SPLINE
SPL {X  -140.879, Y  +291.363, Z    +0.000, E1   +48.273, E3 +172222.912}
SPL {X  -158.845, Y  +331.507, Z    +0.000, E1   +33.834, E3 +172232.246}
SPL {X  -164.164, Y  +356.358, Z    +0.000, E1   +18.707, E3 +172228.569}
SPL {X  -165.341, Y  +368.384, Z    +0.000, E1   +10.076, E3 +172229.313}
SPL {X  -165.648, Y  +377.641, Z    +0.000, E1    +2.653, E3 +172228.664}
SPL {X  -165.650, Y  +380.939, Z    +0.000, E1    -0.407, E3 +172227.475}
SPL {X  -165.650, Y  +384.595, Z    +0.000, E1    -6.546, E3 +172226.958}
SPL {X  -165.650, Y  +389.276, Z    +0.000, E1   -15.245, E3 +172226.466}
SPL {X  -165.650, Y  +395.801, Z    +0.000, E1   -28.236, E3 +172226.094}
SPL {X  -165.650, Y  +403.802, Z    +0.000, E1   -41.748, E3 +172225.915}
SPL {X  -165.650, Y  +419.045, Z    +0.000, E1   -60.641, E3 +172223.236}
SPL {X  -165.650, Y  +474.102, Z    +0.000, E1   -73.446, E3 +172235.019}
SPL {X  -165.650, Y  +637.039, Z    +0.000, E1   -73.842, E3 +172308.092}
ENDSPLINE

SPLINE
SPL {X  -165.650, Y  +617.598, Z    +0.000, E1   -69.273, E3 +172335.159}
ENDSPLINE

SPLINE
SPL {X  -165.650, Y  +623.643, Z    +0.000, E1   -68.543, E3 +172346.326}
SPL {X  -165.650, Y  +635.985, Z    +0.000, E1   -68.274, E3 +172358.704}
SPL {X  -165.650, Y  +656.072, Z    +0.000, E1   -68.403, E3 +172373.999}
SPL {X  -165.650, Y  +669.180, Z    +0.000, E1   -68.170, E3 +172386.465}
SPL {X  -165.417, Y  +684.287, Z    +0.000, E1   -68.467, E3 +172396.261}
SPL {X  -164.268, Y  +696.853, Z    +0.000, E1   -68.071, E3 +172409.890}
SPL {X  -162.443, Y  +707.938, Z    +0.000, E1   -67.853, E3 +172420.624}
SPL {X  -159.812, Y  +719.091, Z    +0.000, E1   -67.711, E3 +172430.930}
SPL {X  -156.969, Y  +728.420, Z    +0.000, E1   -67.278, E3 +172441.712}
SPL {X  -154.751, Y  +734.593, Z    +0.000, E1   -66.864, E3 +172449.693}
SPL {X  -151.443, Y  +742.618, Z    +0.000, E1   -66.527, E3 +172458.688}
SPL {X  -148.198, Y  +749.508, Z    +0.000, E1   -66.065, E3 +172467.169}
SPL {X  -144.642, Y  +756.238, Z    +0.000, E1   -65.678, E3 +172475.035}
SPL {X  -141.719, Y  +761.265, Z    +0.000, E1   -65.117, E3 +172482.168}
SPL {X  -139.420, Y  +764.954, Z    +0.000, E1   -64.577, E3 +172488.031}
SPL {X  -135.180, Y  +771.240, Z    +0.000, E1   -64.104, E3 +172495.561}
SPL {X  -125.028, Y  +784.164, Z    +0.000, E1   -66.760, E3 +172494.031}
SPL {X   -74.840, Y  +823.280, Z    +0.000, E1   -57.857, E3 +172594.563}
SPL {X   -70.065, Y  +825.603, Z    +0.000, E1   -55.379, E3 +172654.865}
ENDSPLINE

SPLINE
SPL {X  -127.072, Y  +781.767, Z    +0.000, E1   -54.186, E3 +172784.068}
SPL {X  -150.680, Y  +744.314, Z    +0.000, E1   -44.608, E3 +172795.024}
SPL {X  -160.361, Y  +717.026, Z    +0.000, E1   -30.396, E3 +172783.878}
SPL {X  -163.361, Y  +702.946, Z    +0.000, E1   -22.646, E3 +172788.997}
SPL {X  -165.092, Y  +689.091, Z    +0.000, E1   -12.938, E3 +172788.567}
SPL {X  -165.629, Y  +678.122, Z    +0.000, E1    -4.178, E3 +172787.714}
SPL {X  -165.650, Y  +673.539, Z    +0.000, E1    -0.057, E3 +172786.811}
SPL {X  -165.650, Y  +671.359, Z    +0.000, E1    +3.116, E3 +172786.168}
SPL {X  -165.650, Y  +667.465, Z    +0.000, E1   +10.413, E3 +172785.962}
SPL {X  -165.650, Y  +662.220, Z    +0.000, E1   +20.600, E3 +172785.654}
SPL {X  -165.650, Y  +652.464, Z    +0.000, E1   +39.379, E3 +172784.602}
SPL {X  -165.650, Y  +636.657, Z    +0.000, E1   +60.410, E3 +172781.890}
SPL {X  -165.650, Y  +613.310, Z    +0.000, E1   +72.038, E3 +172782.249}
SPL {X  -165.650, Y  +568.914, Z    +0.000, E1   +74.438, E3 +172796.834}
SPL {X  -165.650, Y  +420.321, Z    +0.000, E1   +71.570, E3 +172885.488}
ENDSPLINE

SPLINE
SPL {X  -165.650, Y  +437.633, Z    +0.000, E1   +68.421, E3 +172901.236}
ENDSPLINE

SPLINE
SPL {X  -164.513, Y  +359.128, Z    +0.000, E1   +73.170, E3 +172911.470}
SPL {X  -163.967, Y  +354.944, Z    +0.000, E1   +72.327, E3 +172922.823}
SPL {X  -163.372, Y  +351.124, Z    +0.000, E1   +71.295, E3 +172935.415}
SPL {X  -162.653, Y  +347.134, Z    +0.000, E1   +70.371, E3 +172946.650}
SPL {X  -161.430, Y  +341.349, Z    +0.000, E1   +69.492, E3 +172958.725}
SPL {X  -160.389, Y  +337.084, Z    +0.000, E1   +68.301, E3 +172971.812}
SPL {X  -158.795, Y  +331.340, Z    +0.000, E1   +67.291, E3 +172984.498}
SPL {X  -155.058, Y  +320.218, Z    +0.000, E1   +66.982, E3 +172995.804}
SPL {X  -151.047, Y  +310.495, Z    +0.000, E1   +66.593, E3 +173006.438}
SPL {X  -148.187, Y  +304.469, Z    +0.000, E1   +66.029, E3 +173014.817}
SPL {X  -145.703, Y  +299.692, Z    +0.000, E1   +65.663, E3 +173020.983}
SPL {X  -142.469, Y  +293.987, Z    +0.000, E1   +65.133, E3 +173028.696}
SPL {X  -139.022, Y  +288.429, Z    +0.000, E1   +64.807, E3 +173034.894}
SPL {X  -136.717, Y  +284.968, Z    +0.000, E1   +64.044, E3 +173041.487}
SPL {X  -133.061, Y  +279.835, Z    +0.000, E1   +64.204, E3 +173044.900}
SPL {X  -118.927, Y  +263.191, Z    +0.000, E1   +67.951, E3 +173040.913}
SPL {X   -75.220, Y  +230.913, Z    +0.000, E1   +55.539, E3 +173181.544}
ENDSPLINE

SPLINE
SPL {X   -78.274, Y  +232.510, Z    +0.000, E1   +54.798, E3 +173232.027}
SPL {X  -140.879, Y  +291.363, Z    +0.000, E1   +48.273, E3 +173326.360}
SPL {X  -155.054, Y  +320.205, Z    +0.000, E1   +39.591, E3 +173338.811}
SPL {X  -160.978, Y  +339.437, Z    +0.000, E1   +29.257, E3 +173333.441}
SPL {X  -164.164, Y  +356.358, Z    +0.000, E1   +18.707, E3 +173332.017}
SPL {X  -165.519, Y  +371.910, Z    +0.000, E1    +7.409, E3 +173332.426}
SPL {X  -165.650, Y  +380.329, Z    +0.000, E1    +0.239, E3 +173331.272}
SPL {X  -165.650, Y  +381.694, Z    +0.000, E1    -1.679, E3 +173330.544}
SPL {X  -165.650, Y  +384.595, Z    +0.000, E1    -6.546, E3 +173330.406}
SPL {X  -165.650, Y  +389.276, Z    +0.000, E1   -15.245, E3 +173329.915}
SPL {X  -165.650, Y  +395.801, Z    +0.000, E1   -28.236, E3 +173329.542}
SPL {X  -165.650, Y  +403.802, Z    +0.000, E1   -41.748, E3 +173329.363}
SPL {X  -165.650, Y  +419.045, Z    +0.000, E1   -60.641, E3 +173326.684}
SPL {X  -165.650, Y  +474.102, Z    +0.000, E1   -73.446, E3 +173338.467}
SPL {X  -165.650, Y  +640.142, Z    +0.000, E1   -72.635, E3 +173423.752}
ENDSPLINE

SPLINE
SPL {X  -165.650, Y  +619.423, Z    +0.000, E1   -68.618, E3 +173445.949}
ENDSPLINE

SPLINE
SPL {X  -165.650, Y  +635.985, Z    +0.000, E1   -68.274, E3 +173462.152}
SPL {X  -165.650, Y  +647.687, Z    +0.000, E1   -68.151, E3 +173472.652}
SPL {X  -165.650, Y  +665.917, Z    +0.000, E1   -68.414, E3 +173485.412}
SPL {X  -165.417, Y  +684.287, Z    +0.000, E1   -68.467, E3 +173499.709}
SPL {X  -164.268, Y  +696.853, Z    +0.000, E1   -68.071, E3 +173513.338}
SPL {X  -161.478, Y  +712.444, Z    +0.000, E1   -67.895, E3 +173527.545}
SPL {X  -157.774, Y  +725.970, Z    +0.000, E1   -67.383, E3 +173542.547}
SPL {X  -153.458, Y  +737.875, Z    +0.000, E1   -66.902, E3 +173555.622}
SPL {X  -149.433, Y  +746.982, Z    +0.000, E1   -66.131, E3 +173568.253}
SPL {X  -144.642, Y  +756.238, Z    +0.000, E1   -65.678, E3 +173578.483}
SPL {X  -141.719, Y  +761.265, Z    +0.000, E1   -65.117, E3 +173585.616}
SPL {X  -139.420, Y  +764.954, Z    +0.000, E1   -64.577, E3 +173591.480}
SPL {X  -136.483, Y  +769.374, Z    +0.000, E1   -64.163, E3 +173597.135}
SPL {X  -133.523, Y  +773.539, Z    +0.000, E1   -63.962, E3 +173601.403}
SPL {X  -125.028, Y  +784.164, Z    +0.000, E1   -66.760, E3 +173597.479}
SPL {X   -71.589, Y  +824.882, Z    +0.000, E1   -56.415, E3 +173724.544}
ENDSPLINE

SPLINE
SPL {X  -127.072, Y  +781.767, Z    +0.000, E1   -54.186, E3 +173887.516}
SPL {X  -150.680, Y  +744.314, Z    +0.000, E1   -44.608, E3 +173898.472}
SPL {X  -160.361, Y  +717.026, Z    +0.000, E1   -30.396, E3 +173887.326}
SPL {X  -163.361, Y  +702.946, Z    +0.000, E1   -22.646, E3 +173892.445}
SPL {X  -165.092, Y  +689.091, Z    +0.000, E1   -12.938, E3 +173892.015}
SPL {X  -165.569, Y  +680.695, Z    +0.000, E1    -6.245, E3 +173890.700}
SPL {X  -165.650, Y  +673.489, Z    +0.000, E1    -0.162, E3 +173890.204}
SPL {X  -165.650, Y  +669.039, Z    +0.000, E1    +7.218, E3 +173889.465}
SPL {X  -165.650, Y  +662.220, Z    +0.000, E1   +20.600, E3 +173889.103}
SPL {X  -165.650, Y  +652.464, Z    +0.000, E1   +39.379, E3 +173888.050}
SPL {X  -165.650, Y  +634.871, Z    +0.000, E1   +61.762, E3 +173885.283}
SPL {X  -165.650, Y  +574.769, Z    +0.000, E1   +74.441, E3 +173897.931}
SPL {X  -165.650, Y  +420.321, Z    +0.000, E1   +71.570, E3 +173988.936}
ENDSPLINE

SPLINE
SPL {X  -165.650, Y  +437.633, Z    +0.000, E1   +68.421, E3 +174004.684}
ENDSPLINE

SPLINE
SPL {X  -164.513, Y  +359.128, Z    +0.000, E1   +73.170, E3 +174014.918}
SPL {X  -163.967, Y  +354.944, Z    +0.000, E1   +72.327, E3 +174026.271}
SPL {X  -163.372, Y  +351.124, Z    +0.000, E1   +71.295, E3 +174038.863}
SPL {X  -162.653, Y  +347.134, Z    +0.000, E1   +70.371, E3 +174050.099}
SPL {X  -161.430, Y  +341.349, Z    +0.000, E1   +69.492, E3 +174062.173}
SPL {X  -160.389, Y  +337.084, Z    +0.000, E1   +68.301, E3 +174075.260}
SPL {X  -158.795, Y  +331.340, Z    +0.000, E1   +67.291, E3 +174087.947}
SPL {X  -155.058, Y  +320.218, Z    +0.000, E1   +66.982, E3 +174099.253}
SPL {X  -151.047, Y  +310.495, Z    +0.000, E1   +66.593, E3 +174109.886}
SPL {X  -146.639, Y  +301.448, Z    +0.000, E1   +65.839, E3 +174122.095}
SPL {X  -142.469, Y  +293.987, Z    +0.000, E1   +65.133, E3 +174132.144}
SPL {X  -139.022, Y  +288.429, Z    +0.000, E1   +64.807, E3 +174138.343}
SPL {X  -136.717, Y  +284.968, Z    +0.000, E1   +64.044, E3 +174144.935}
SPL {X  -133.061, Y  +279.835, Z    +0.000, E1   +64.204, E3 +174148.349}
SPL {X  -118.927, Y  +263.191, Z    +0.000, E1   +67.951, E3 +174144.361}
SPL {X   -76.819, Y  +231.739, Z    +0.000, E1   +54.834, E3 +174322.367}
ENDSPLINE

SPLINE
SPL {X  -140.879, Y  +291.363, Z    +0.000, E1   +48.273, E3 +174429.808}
SPL {X  -158.845, Y  +331.507, Z    +0.000, E1   +33.834, E3 +174439.143}
SPL {X  -164.164, Y  +356.358, Z    +0.000, E1   +18.707, E3 +174435.466}
SPL {X  -165.341, Y  +368.384, Z    +0.000, E1   +10.076, E3 +174436.210}
SPL {X  -165.648, Y  +377.641, Z    +0.000, E1    +2.653, E3 +174435.561}
SPL {X  -165.650, Y  +380.939, Z    +0.000, E1    -0.407, E3 +174434.371}
SPL {X  -165.650, Y  +385.900, Z    +0.000, E1    -8.711, E3 +174433.816}
SPL {X  -165.650, Y  +390.854, Z    +0.000, E1   -18.692, E3 +174432.991}
SPL {X  -165.650, Y  +395.801, Z    +0.000, E1   -28.236, E3 +174432.990}
SPL {X  -165.650, Y  +403.802, Z    +0.000, E1   -41.748, E3 +174432.811}
SPL {X  -165.650, Y  +418.088, Z    +0.000, E1   -59.974, E3 +174430.084}
SPL {X  -165.650, Y  +461.994, Z    +0.000, E1   -72.657, E3 +174438.222}
SPL {X  -165.650, Y  +492.072, Z    +0.000, E1   -73.925, E3 +174448.324}
SPL {X  -165.650, Y  +640.142, Z    +0.000, E1   -72.635, E3 +174527.200}
ENDSPLINE

SPLINE
SPL {X  -165.650, Y  +612.217, Z    +0.000, E1   -68.647, E3 +174543.125}
ENDSPLINE

SPLINE
SPL {X  -165.650, Y  +623.643, Z    +0.000, E1   -68.543, E3 +174553.222}
SPL {X  -165.650, Y  +635.985, Z    +0.000, E1   -68.274, E3 +174565.601}
SPL {X  -165.650, Y  +647.687, Z    +0.000, E1   -68.151, E3 +174576.100}
SPL {X  -165.650, Y  +665.917, Z    +0.000, E1   -68.414, E3 +174588.860}
SPL {X  -165.417, Y  +684.287, Z    +0.000, E1   -68.467, E3 +174603.157}
SPL {X  -164.655, Y  +693.631, Z    +0.000, E1   -68.130, E3 +174613.508}
SPL {X  -162.986, Y  +705.089, Z    +0.000, E1   -67.915, E3 +174624.827}
SPL {X  -160.378, Y  +716.957, Z    +0.000, E1   -67.874, E3 +174634.647}
SPL {X  -157.774, Y  +725.970, Z    +0.000, E1   -67.383, E3 +174645.995}
SPL {X  -153.458, Y  +737.875, Z    +0.000, E1   -66.902, E3 +174659.070}
SPL {X  -150.971, Y  +743.674, Z    +0.000, E1   -66.152, E3 +174668.728}
SPL {X  -148.198, Y  +749.508, Z    +0.000, E1   -66.065, E3 +174674.065}
SPL {X  -144.642, Y  +756.238, Z    +0.000, E1   -65.678, E3 +174681.932}
SPL {X  -140.398, Y  +763.411, Z    +0.000, E1   -64.853, E3 +174692.408}
SPL {X  -136.483, Y  +769.374, Z    +0.000, E1   -64.163, E3 +174700.583}
SPL {X  -133.523, Y  +773.539, Z    +0.000, E1   -63.962, E3 +174704.852}
SPL {X  -127.756, Y  +780.943, Z    +0.000, E1   -66.344, E3 +174700.446}
SPL {X  -118.855, Y  +790.884, Z    +0.000, E1   -67.633, E3 +174701.815}
SPL {X   -74.840, Y  +823.280, Z    +0.000, E1   -57.857, E3 +174801.460}
SPL {X   -70.065, Y  +825.603, Z    +0.000, E1   -55.379, E3 +174861.762}
ENDSPLINE

SPLINE
SPL {X  -127.072, Y  +781.767, Z    +0.000, E1   -54.186, E3 +174990.964}
SPL {X  -150.680, Y  +744.314, Z    +0.000, E1   -44.608, E3 +175001.921}
SPL {X  -162.376, Y  +708.273, Z    +0.000, E1   -25.870, E3 +174994.044}
SPL {X  -165.092, Y  +689.091, Z    +0.000, E1   -12.938, E3 +174995.463}
SPL {X  -165.569, Y  +680.695, Z    +0.000, E1    -6.245, E3 +174994.148}
SPL {X  -165.650, Y  +673.489, Z    +0.000, E1    -0.162, E3 +174993.653}
SPL {X  -165.650, Y  +669.039, Z    +0.000, E1    +7.218, E3 +174992.914}
SPL {X  -165.650, Y  +663.739, Z    +0.000, E1   +17.756, E3 +174992.605}
SPL {X  -165.650, Y  +656.188, Z    +0.000, E1   +32.567, E3 +174991.886}
SPL {X  -165.650, Y  +648.712, Z    +0.000, E1   +45.195, E3 +174991.509}
SPL {X  -165.650, Y  +634.871, Z    +0.000, E1   +61.762, E3 +174988.731}
SPL {X  -165.650, Y  +574.769, Z    +0.000, E1   +74.441, E3 +175001.379}
SPL {X  -165.650, Y  +420.321, Z    +0.000, E1   +71.570, E3 +175092.384}
ENDSPLINE

SPLINE
SPL {X  -165.650, Y  +437.633, Z    +0.000, E1   +68.421, E3 +175108.133}
ENDSPLINE

SPLINE
SPL {X  -164.513, Y  +359.128, Z    +0.000, E1   +73.170, E3 +175118.366}
SPL {X  -163.967, Y  +354.944, Z    +0.000, E1   +72.327, E3 +175129.719}
SPL {X  -163.372, Y  +351.124, Z    +0.000, E1   +71.295, E3 +175142.312}
SPL {X  -162.653, Y  +347.134, Z    +0.000, E1   +70.371, E3 +175153.547}
SPL {X  -161.451, Y  +341.438, Z    +0.000, E1   +69.889, E3 +175161.866}
SPL {X  -161.195, Y  +340.340, Z    +0.000, E1   +68.690, E3 +175173.087}
SPL {X  -159.328, Y  +333.173, Z    +0.000, E1   +67.752, E3 +175186.308}
SPL {X  -157.072, Y  +325.885, Z    +0.000, E1   +67.020, E3 +175197.717}
SPL {X  -153.570, Y  +316.402, Z    +0.000, E1   +66.799, E3 +175207.079}
SPL {X  -149.308, Y  +306.758, Z    +0.000, E1   +66.321, E3 +175218.205}
SPL {X  -145.703, Y  +299.692, Z    +0.000, E1   +65.663, E3 +175227.880}
SPL {X  -142.469, Y  +293.987, Z    +0.000, E1   +65.133, E3 +175235.592}
SPL {X  -139.022, Y  +288.429, Z    +0.000, E1   +64.807, E3 +175241.791}
SPL {X  -136.717, Y  +284.968, Z    +0.000, E1   +64.044, E3 +175248.383}
SPL {X  -133.061, Y  +279.835, Z    +0.000, E1   +64.204, E3 +175251.797}
SPL {X  -118.927, Y  +263.191, Z    +0.000, E1   +67.951, E3 +175247.809}
SPL {X   -75.220, Y  +230.913, Z    +0.000, E1   +55.539, E3 +175388.441}
ENDSPLINE

SPLINE
SPL {X   -78.274, Y  +232.510, Z    +0.000, E1   +54.798, E3 +175438.923}
SPL {X  -140.879, Y  +291.363, Z    +0.000, E1   +48.273, E3 +175533.257}
SPL {X  -158.845, Y  +331.507, Z    +0.000, E1   +33.834, E3 +175542.591}
SPL {X  -164.164, Y  +356.358, Z    +0.000, E1   +18.707, E3 +175538.914}
SPL {X  -165.519, Y  +371.910, Z    +0.000, E1    +7.409, E3 +175539.323}
SPL {X  -165.650, Y  +380.329, Z    +0.000, E1    +0.239, E3 +175538.169}
SPL {X  -165.650, Y  +381.694, Z    +0.000, E1    -1.679, E3 +175537.441}
SPL {X  -165.650, Y  +385.900, Z    +0.000, E1    -8.711, E3 +175537.264}
SPL {X  -165.650, Y  +390.854, Z    +0.000, E1   -18.692, E3 +175536.440}
SPL {X  -165.650, Y  +395.801, Z    +0.000, E1   -28.236, E3 +175536.439}
SPL {X  -165.650, Y  +403.802, Z    +0.000, E1   -41.748, E3 +175536.259}
SPL {X  -165.650, Y  +419.045, Z    +0.000, E1   -60.641, E3 +175533.581}
SPL {X  -165.650, Y  +474.102, Z    +0.000, E1   -73.446, E3 +175545.364}
SPL {X  -165.650, Y  +640.142, Z    +0.000, E1   -72.635, E3 +175630.648}
ENDSPLINE

SPLINE
SPL {X  -165.650, Y  +612.217, Z    +0.000, E1   -68.647, E3 +175646.574}
ENDSPLINE

SPLINE
SPL {X  -165.650, Y  +623.643, Z    +0.000, E1   -68.543, E3 +175656.670}
SPL {X  -165.650, Y  +635.985, Z    +0.000, E1   -68.274, E3 +175669.049}
SPL {X  -165.650, Y  +656.072, Z    +0.000, E1   -68.403, E3 +175684.343}
SPL {X  -165.650, Y  +669.180, Z    +0.000, E1   -68.170, E3 +175696.810}
SPL {X  -165.417, Y  +684.287, Z    +0.000, E1   -68.467, E3 +175706.605}
SPL {X  -164.268, Y  +696.853, Z    +0.000, E1   -68.071, E3 +175720.235}
SPL {X  -162.443, Y  +707.938, Z    +0.000, E1   -67.853, E3 +175730.969}
SPL {X  -159.812, Y  +719.091, Z    +0.000, E1   -67.711, E3 +175741.275}
SPL {X  -156.969, Y  +728.420, Z    +0.000, E1   -67.278, E3 +175752.057}
SPL {X  -154.751, Y  +734.593, Z    +0.000, E1   -66.864, E3 +175760.038}
SPL {X  -151.443, Y  +742.618, Z    +0.000, E1   -66.527, E3 +175769.033}
SPL {X  -146.969, Y  +751.920, Z    +0.000, E1   -66.066, E3 +175779.529}
SPL {X  -142.811, Y  +759.434, Z    +0.000, E1   -65.254, E3 +175790.378}
SPL {X  -139.420, Y  +764.954, Z    +0.000, E1   -64.577, E3 +175798.376}
SPL {X  -136.483, Y  +769.374, Z    +0.000, E1   -64.163, E3 +175804.031}
SPL {X  -133.523, Y  +773.539, Z    +0.000, E1   -63.962, E3 +175808.300}
SPL {X  -125.028, Y  +784.164, Z    +0.000, E1   -66.760, E3 +175804.375}
SPL {X   -71.589, Y  +824.882, Z    +0.000, E1   -56.415, E3 +175931.440}
ENDSPLINE

SPLINE
SPL {X  -127.072, Y  +781.767, Z    +0.000, E1   -54.186, E3 +176094.412}
SPL {X  -150.680, Y  +744.314, Z    +0.000, E1   -44.608, E3 +176105.369}
SPL {X  -160.361, Y  +717.026, Z    +0.000, E1   -30.396, E3 +176094.223}
SPL {X  -163.361, Y  +702.946, Z    +0.000, E1   -22.646, E3 +176099.342}
SPL {X  -165.092, Y  +689.091, Z    +0.000, E1   -12.938, E3 +176098.911}
SPL {X  -165.629, Y  +678.122, Z    +0.000, E1    -4.178, E3 +176098.058}
SPL {X  -165.650, Y  +673.539, Z    +0.000, E1    -0.057, E3 +176097.156}
SPL {X  -165.650, Y  +671.359, Z    +0.000, E1    +3.116, E3 +176096.513}
SPL {X  -165.650, Y  +667.465, Z    +0.000, E1   +10.413, E3 +176096.307}
SPL {X  -165.650, Y  +662.220, Z    +0.000, E1   +20.600, E3 +176095.999}
SPL {X  -165.650, Y  +652.464, Z    +0.000, E1   +39.379, E3 +176094.947}
SPL {X  -165.650, Y  +636.657, Z    +0.000, E1   +60.410, E3 +176092.235}
SPL {X  -165.650, Y  +613.310, Z    +0.000, E1   +72.038, E3 +176092.594}
SPL {X  -165.650, Y  +568.914, Z    +0.000, E1   +74.438, E3 +176107.179}
SPL {X  -165.650, Y  +420.321, Z    +0.000, E1   +71.570, E3 +176195.832}
ENDSPLINE

SPLINE
SPL {X  -165.650, Y  +437.633, Z    +0.000, E1   +68.421, E3 +176211.581}
ENDSPLINE

SPLINE
SPL {X  -164.513, Y  +359.128, Z    +0.000, E1   +73.170, E3 +176221.814}
SPL {X  -163.967, Y  +354.944, Z    +0.000, E1   +72.327, E3 +176233.168}
SPL {X  -163.372, Y  +351.124, Z    +0.000, E1   +71.295, E3 +176245.760}
SPL {X  -162.653, Y  +347.134, Z    +0.000, E1   +70.371, E3 +176256.995}
SPL {X  -161.430, Y  +341.349, Z    +0.000, E1   +69.492, E3 +176269.069}
SPL {X  -160.389, Y  +337.084, Z    +0.000, E1   +68.301, E3 +176282.157}
SPL {X  -159.245, Y  +332.881, Z    +0.000, E1   +67.496, E3 +176291.816}
SPL {X  -157.072, Y  +325.885, Z    +0.000, E1   +67.020, E3 +176301.166}
SPL {X  -154.432, Y  +318.577, Z    +0.000, E1   +66.843, E3 +176308.371}
SPL {X  -151.047, Y  +310.495, Z    +0.000, E1   +66.593, E3 +176316.783}
SPL {X  -146.639, Y  +301.448, Z    +0.000, E1   +65.839, E3 +176328.992}
SPL {X  -142.469, Y  +293.987, Z    +0.000, E1   +65.133, E3 +176339.041}
SPL {X  -139.022, Y  +288.429, Z    +0.000, E1   +64.807, E3 +176345.239}
SPL {X  -136.717, Y  +284.968, Z    +0.000, E1   +64.044, E3 +176351.831}
SPL {X  -133.061, Y  +279.835, Z    +0.000, E1   +64.204, E3 +176355.245}
SPL {X  -118.927, Y  +263.191, Z    +0.000, E1   +67.951, E3 +176351.258}
SPL {X   -76.819, Y  +231.739, Z    +0.000, E1   +54.834, E3 +176529.264}
ENDSPLINE

SPLINE
SPL {X  -140.879, Y  +291.363, Z    +0.000, E1   +48.273, E3 +176636.705}
SPL {X  -158.845, Y  +331.507, Z    +0.000, E1   +33.834, E3 +176646.040}
SPL {X  -164.164, Y  +356.358, Z    +0.000, E1   +18.707, E3 +176642.362}
SPL {X  -165.341, Y  +368.384, Z    +0.000, E1   +10.076, E3 +176643.106}
SPL {X  -165.648, Y  +377.641, Z    +0.000, E1    +2.653, E3 +176642.457}
SPL {X  -165.650, Y  +380.500, Z    +0.000, E1    -0.000, E3 +176641.488}
SPL {X  -165.650, Y  +381.694, Z    +0.000, E1    -1.679, E3 +176640.889}
SPL {X  -165.650, Y  +384.595, Z    +0.000, E1    -6.546, E3 +176640.751}
SPL {X  -165.650, Y  +389.276, Z    +0.000, E1   -15.245, E3 +176640.259}
SPL {X  -165.650, Y  +395.801, Z    +0.000, E1   -28.236, E3 +176639.887}
SPL {X  -165.650, Y  +403.802, Z    +0.000, E1   -41.748, E3 +176639.708}
SPL {X  -165.650, Y  +419.045, Z    +0.000, E1   -60.641, E3 +176637.029}
SPL {X  -165.650, Y  +474.102, Z    +0.000, E1   -73.446, E3 +176648.812}
SPL {X  -165.650, Y  +640.142, Z    +0.000, E1   -72.635, E3 +176734.097}
ENDSPLINE

SPLINE
SPL {X  -165.650, Y  +619.423, Z    +0.000, E1   -68.618, E3 +176756.294}
ENDSPLINE

SPLINE
SPL {X  -165.650, Y  +635.985, Z    +0.000, E1   -68.274, E3 +176772.497}
SPL {X  -165.650, Y  +647.687, Z    +0.000, E1   -68.151, E3 +176782.997}
SPL {X  -165.650, Y  +665.917, Z    +0.000, E1   -68.414, E3 +176795.756}
SPL {X  -165.417, Y  +684.287, Z    +0.000, E1   -68.467, E3 +176810.054}
SPL {X  -164.268, Y  +696.853, Z    +0.000, E1   -68.071, E3 +176823.683}
SPL {X  -161.478, Y  +712.444, Z    +0.000, E1   -67.895, E3 +176837.890}
SPL {X  -157.774, Y  +725.970, Z    +0.000, E1   -67.383, E3 +176852.891}
SPL {X  -154.751, Y  +734.593, Z    +0.000, E1   -66.864, E3 +176863.486}
SPL {X  -151.443, Y  +742.618, Z    +0.000, E1   -66.527, E3 +176872.481}
SPL {X  -146.969, Y  +751.920, Z    +0.000, E1   -66.066, E3 +176882.978}
SPL {X  -142.811, Y  +759.434, Z    +0.000, E1   -65.254, E3 +176893.826}
SPL {X  -139.420, Y  +764.954, Z    +0.000, E1   -64.577, E3 +176901.825}
SPL {X  -136.483, Y  +769.374, Z    +0.000, E1   -64.163, E3 +176907.480}
SPL {X  -133.523, Y  +773.539, Z    +0.000, E1   -63.962, E3 +176911.748}
SPL {X  -125.028, Y  +784.164, Z    +0.000, E1   -66.760, E3 +176907.824}
SPL {X   -71.589, Y  +824.882, Z    +0.000, E1   -56.415, E3 +177034.889}
ENDSPLINE

SPLINE
SPL {X  -127.072, Y  +781.767, Z    +0.000, E1   -54.186, E3 +177197.861}
SPL {X  -150.680, Y  +744.314, Z    +0.000, E1   -44.608, E3 +177208.817}
SPL {X  -162.376, Y  +708.273, Z    +0.000, E1   -25.870, E3 +177200.941}
SPL {X  -165.092, Y  +689.091, Z    +0.000, E1   -12.938, E3 +177202.360}
SPL {X  -165.629, Y  +678.122, Z    +0.000, E1    -4.178, E3 +177201.507}
SPL {X  -165.650, Y  +673.539, Z    +0.000, E1    -0.057, E3 +177200.604}
SPL {X  -165.650, Y  +671.359, Z    +0.000, E1    +3.116, E3 +177199.961}
SPL {X  -165.650, Y  +665.277, Z    +0.000, E1   +14.409, E3 +177199.606}
SPL {X  -165.650, Y  +659.573, Z    +0.000, E1   +26.182, E3 +177199.354}
SPL {X  -165.650, Y  +652.464, Z    +0.000, E1   +39.379, E3 +177198.395}
SPL {X  -165.650, Y  +634.871, Z    +0.000, E1   +61.762, E3 +177195.628}
SPL {X  -165.650, Y  +574.769, Z    +0.000, E1   +74.441, E3 +177208.276}
SPL {X  -165.650, Y  +420.321, Z    +0.000, E1   +71.570, E3 +177299.281}
ENDSPLINE

SPLINE
SPL {X  -165.650, Y  +437.633, Z    +0.000, E1   +68.421, E3 +177315.029}
ENDSPLINE

SPLINE
SPL {X  -164.513, Y  +359.128, Z    +0.000, E1   +73.170, E3 +177325.263}
SPL {X  -163.967, Y  +354.944, Z    +0.000, E1   +72.327, E3 +177336.616}
SPL {X  -163.372, Y  +351.124, Z    +0.000, E1   +71.295, E3 +177349.208}
SPL {X  -162.653, Y  +347.134, Z    +0.000, E1   +70.371, E3 +177360.444}
SPL {X  -161.430, Y  +341.349, Z    +0.000, E1   +69.492, E3 +177372.518}
SPL {X  -160.871, Y  +338.999, Z    +0.000, E1   +68.071, E3 +177386.034}
ENDSPLINE

SPLINE
SPL {X  -161.965, Y  +343.754, Z    +0.000, E1   +65.498, E3 +177402.203}
ENDSPLINE

SPLINE
SPL {X  -158.875, Y  +331.610, Z    +0.000, E1   +64.945, E3 +177417.386}
SPL {X  -154.872, Y  +319.724, Z    +0.000, E1   +64.496, E3 +177431.300}
SPL {X  -151.091, Y  +310.592, Z    +0.000, E1   +63.929, E3 +177443.240}
SPL {X  -148.836, Y  +305.783, Z    +0.000, E1   +63.120, E3 +177452.372}
SPL {X  -145.492, Y  +299.305, Z    +0.000, E1   +63.037, E3 +177458.864}
SPL {X  -142.120, Y  +293.401, Z    +0.000, E1   +62.602, E3 +177466.543}
SPL {X  -139.854, Y  +289.726, Z    +0.000, E1   +61.679, E3 +177474.449}
SPL {X  -135.997, Y  +283.923, Z    +0.000, E1   +62.034, E3 +177478.098}
SPL {X  -124.991, Y  +269.793, Z    +0.000, E1   +65.852, E3 +177473.087}
SPL {X   -80.641, Y  +233.804, Z    +0.000, E1   +55.283, E3 +177604.202}
ENDSPLINE

SPLINE
SPL {X  -132.197, Y  +278.681, Z    +0.000, E1   +49.692, E3 +177738.074}
SPL {X  -156.075, Y  +322.998, Z    +0.000, E1   +35.140, E3 +177743.155}
SPL {X  -162.799, Y  +347.901, Z    +0.000, E1   +22.644, E3 +177745.661}
SPL {X  -164.930, Y  +363.071, Z    +0.000, E1   +13.041, E3 +177743.401}
SPL {X  -165.629, Y  +375.893, Z    +0.000, E1    +3.908, E3 +177743.259}
SPL {X  -165.650, Y  +380.596, Z    +0.000, E1    -0.052, E3 +177741.940}
SPL {X  -165.650, Y  +383.460, Z    +0.000, E1    -3.790, E3 +177741.265}
SPL {X  -165.650, Y  +389.311, Z    +0.000, E1   -13.234, E3 +177740.751}
SPL {X  -165.650, Y  +395.103, Z    +0.000, E1   -23.932, E3 +177740.044}
SPL {X  -165.650, Y  +401.925, Z    +0.000, E1   -35.470, E3 +177739.311}
SPL {X  -165.650, Y  +410.900, Z    +0.000, E1   -46.977, E3 +177739.928}
SPL {X  -165.650, Y  +423.066, Z    +0.000, E1   -61.140, E3 +177735.659}
SPL {X  -165.650, Y  +461.121, Z    +0.000, E1   -74.504, E3 +177737.008}
SPL {X  -165.650, Y  +487.674, Z    +0.000, E1   -70.215, E3 +177759.819}
SPL {X  -165.650, Y  +590.449, Z    +0.000, E1   -68.990, E3 +177827.764}
ENDSPLINE

SPLINE
SPL {X  -165.650, Y  +577.071, Z    +0.000, E1   -65.152, E3 +177846.087}
ENDSPLINE

SPLINE
SPL {X  -165.650, Y  +580.077, Z    +0.000, E1   -64.018, E3 +177857.665}
SPL {X  -165.650, Y  +590.532, Z    +0.000, E1   -63.993, E3 +177868.231}
SPL {X  -165.650, Y  +600.616, Z    +0.000, E1   -64.059, E3 +177877.804}
SPL {X  -165.650, Y  +609.299, Z    +0.000, E1   -64.001, E3 +177886.829}
SPL {X  -165.650, Y  +618.778, Z    +0.000, E1   -63.957, E3 +177896.686}
SPL {X  -165.650, Y  +634.916, Z    +0.000, E1   -64.117, E3 +177911.735}
SPL {X  -165.650, Y  +648.710, Z    +0.000, E1   -63.999, E3 +177926.145}
SPL {X  -165.650, Y  +658.618, Z    +0.000, E1   -64.006, E3 +177935.962}
SPL {X  -165.650, Y  +670.604, Z    +0.000, E1   -64.021, E3 +177947.876}
SPL {X  -165.270, Y  +686.708, Z    +0.000, E1   -64.001, E3 +177964.219}
SPL {X  -163.641, Y  +701.218, Z    +0.000, E1   -63.638, E3 +177981.363}
SPL {X  -161.003, Y  +714.463, Z    +0.000, E1   -63.428, E3 +177996.034}
SPL {X  -157.854, Y  +725.721, Z    +0.000, E1   -62.989, E3 +178010.283}
SPL {X  -155.984, Y  +731.258, Z    +0.000, E1   -62.241, E3 +178020.429}
SPL {X  -153.281, Y  +738.308, Z    +0.000, E1   -62.233, E3 +178027.617}
SPL {X  -150.070, Y  +745.636, Z    +0.000, E1   -61.982, E3 +178036.363}
SPL {X  -148.438, Y  +749.026, Z    +0.000, E1   -61.150, E3 +178044.370}
SPL {X  -145.760, Y  +754.202, Z    +0.000, E1   -61.108, E3 +178049.786}
SPL {X  -143.078, Y  +758.979, Z    +0.000, E1   -60.553, E3 +178057.445}
SPL {X  -139.815, Y  +764.336, Z    +0.000, E1   -60.025, E3 +178065.297}
SPL {X  -130.672, Y  +777.307, Z    +0.000, E1   -63.098, E3 +178063.588}
SPL {X   -84.123, Y  +818.200, Z    +0.000, E1   -55.499, E3 +178177.101}
ENDSPLINE

SPLINE
SPL {X  -127.502, Y  +781.251, Z    +0.000, E1   -49.821, E3 +178309.234}
SPL {X  -151.617, Y  +742.224, Z    +0.000, E1   -39.442, E3 +178325.817}
SPL {X  -159.277, Y  +721.007, Z    +0.000, E1   -30.118, E3 +178324.994}
SPL {X  -163.701, Y  +700.836, Z    +0.000, E1   -18.960, E3 +178321.709}
SPL {X  -165.229, Y  +687.300, Z    +0.000, E1   -10.302, E3 +178321.664}
SPL {X  -165.592, Y  +679.896, Z    +0.000, E1    -5.071, E3 +178320.945}
SPL {X  -165.650, Y  +674.350, Z    +0.000, E1    -0.828, E3 +178320.319}
SPL {X  -165.650, Y  +672.653, Z    +0.000, E1    +0.827, E3 +178319.512}
SPL {X  -165.650, Y  +668.094, Z    +0.000, E1    +7.098, E3 +178318.881}
SPL {X  -165.650, Y  +662.291, Z    +0.000, E1   +16.729, E3 +178318.807}
SPL {X  -165.650, Y  +656.382, Z    +0.000, E1   +26.732, E3 +178318.365}
SPL {X  -165.650, Y  +648.240, Z    +0.000, E1   +42.276, E3 +178313.799}
SPL {X  -165.650, Y  +638.782, Z    +0.000, E1   +47.719, E3 +178321.009}
SPL {X  -165.650, Y  +622.329, Z    +0.000, E1   +68.753, E3 +178308.548}
SPL {X  -165.650, Y  +589.967, Z    +0.000, E1   +71.395, E3 +178321.174}
SPL {X  -165.650, Y  +573.012, Z    +0.000, E1   +68.475, E3 +178337.386}
SPL {X  -165.650, Y  +459.505, Z    +0.000, E1   +68.780, E3 +178409.110}
ENDSPLINE

SPLINE
SPL {X  -165.650, Y  +483.715, Z    +0.000, E1   +63.891, E3 +178425.404}
ENDSPLINE

SPLINE
SPL {X  -165.650, Y  +474.626, Z    +0.000, E1   +63.707, E3 +178435.933}
SPL {X  -165.650, Y  +465.190, Z    +0.000, E1   +63.660, E3 +178445.788}
SPL {X  -165.650, Y  +456.011, Z    +0.000, E1   +63.585, E3 +178455.683}
SPL {X  -165.650, Y  +441.325, Z    +0.000, E1   +63.847, E3 +178468.652}
SPL {X  -165.552, Y  +372.799, Z    +0.000, E1   +69.633, E3 +178481.058}
SPL {X  -165.443, Y  +370.231, Z    +0.000, E1   +68.724, E3 +178490.988}
SPL {X  -164.776, Y  +361.504, Z    +0.000, E1   +68.225, E3 +178502.462}
SPL {X  -164.241, Y  +356.944, Z    +0.000, E1   +66.930, E3 +178516.985}
SPL {X  -163.312, Y  +350.765, Z    +0.000, E1   +66.182, E3 +178528.162}
SPL {X  -163.046, Y  +349.241, Z    +0.000, E1   +65.245, E3 +178536.734}
SPL {X  -160.229, Y  +336.468, Z    +0.000, E1   +65.236, E3 +178548.717}
SPL {X  -157.078, Y  +325.903, Z    +0.000, E1   +64.692, E3 +178562.163}
SPL {X  -153.279, Y  +315.688, Z    +0.000, E1   +64.219, E3 +178574.736}
SPL {X  -149.447, Y  +307.046, Z    +0.000, E1   +63.460, E3 +178587.321}
SPL {X  -145.492, Y  +299.305, Z    +0.000, E1   +63.037, E3 +178596.795}
SPL {X  -142.120, Y  +293.401, Z    +0.000, E1   +62.602, E3 +178604.474}
SPL {X  -139.854, Y  +289.726, Z    +0.000, E1   +61.679, E3 +178612.380}
SPL {X  -135.997, Y  +283.923, Z    +0.000, E1   +62.034, E3 +178616.029}
SPL {X  -124.991, Y  +269.793, Z    +0.000, E1   +65.852, E3 +178611.018}
SPL {X   -80.641, Y  +233.804, Z    +0.000, E1   +55.283, E3 +178742.133}
ENDSPLINE

SPLINE
SPL {X  -126.633, Y  +271.710, Z    +0.000, E1   +51.055, E3 +178872.599}
SPL {X  -147.744, Y  +303.590, Z    +0.000, E1   +42.717, E3 +178881.091}
SPL {X  -158.730, Y  +331.121, Z    +0.000, E1   +31.334, E3 +178880.999}
SPL {X  -162.799, Y  +347.901, Z    +0.000, E1   +22.644, E3 +178883.592}
SPL {X  -164.930, Y  +363.071, Z    +0.000, E1   +13.041, E3 +178881.332}
SPL {X  -165.629, Y  +375.893, Z    +0.000, E1    +3.908, E3 +178881.190}
SPL {X  -165.650, Y  +380.596, Z    +0.000, E1    -0.052, E3 +178879.872}
SPL {X  -165.650, Y  +383.460, Z    +0.000, E1    -3.790, E3 +178879.196}
SPL {X  -165.650, Y  +387.326, Z    +0.000, E1   -10.041, E3 +178879.068}
SPL {X  -165.650, Y  +392.519, Z    +0.000, E1   -19.014, E3 +178878.221}
SPL {X  -165.650, Y  +401.925, Z    +0.000, E1   -35.470, E3 +178877.242}
SPL {X  -165.650, Y  +410.900, Z    +0.000, E1   -46.977, E3 +178877.859}
SPL {X  -165.650, Y  +420.865, Z    +0.000, E1   -58.704, E3 +178874.750}
SPL {X  -165.650, Y  +450.181, Z    +0.000, E1   -73.218, E3 +178872.697}
SPL {X  -165.650, Y  +487.674, Z    +0.000, E1   -70.215, E3 +178897.750}
SPL {X  -165.650, Y  +585.482, Z    +0.000, E1   -67.026, E3 +178976.912}
ENDSPLINE

SPLINE
SPL {X  -165.650, Y  +571.836, Z    +0.000, E1   -64.066, E3 +178986.932}
ENDSPLINE

SPLINE
SPL {X  -165.650, Y  +580.077, Z    +0.000, E1   -64.018, E3 +178995.596}
SPL {X  -165.650, Y  +590.532, Z    +0.000, E1   -63.993, E3 +179006.162}
SPL {X  -165.650, Y  +604.471, Z    +0.000, E1   -64.071, E3 +179019.669}
SPL {X  -165.650, Y  +618.778, Z    +0.000, E1   -63.957, E3 +179034.617}
SPL {X  -165.650, Y  +634.916, Z    +0.000, E1   -64.117, E3 +179049.666}
SPL {X  -165.650, Y  +648.710, Z    +0.000, E1   -63.999, E3 +179064.076}
SPL {X  -165.650, Y  +658.618, Z    +0.000, E1   -64.006, E3 +179073.894}
SPL {X  -165.650, Y  +670.604, Z    +0.000, E1   -64.021, E3 +179085.807}
SPL {X  -165.270, Y  +686.708, Z    +0.000, E1   -64.001, E3 +179102.150}
SPL {X  -163.641, Y  +701.218, Z    +0.000, E1   -63.638, E3 +179119.294}
SPL {X  -161.003, Y  +714.463, Z    +0.000, E1   -63.428, E3 +179133.965}
SPL {X  -157.854, Y  +725.721, Z    +0.000, E1   -62.989, E3 +179148.214}
SPL {X  -155.984, Y  +731.258, Z    +0.000, E1   -62.241, E3 +179158.360}
SPL {X  -153.281, Y  +738.308, Z    +0.000, E1   -62.233, E3 +179165.548}
SPL {X  -150.070, Y  +745.636, Z    +0.000, E1   -61.982, E3 +179174.294}
SPL {X  -148.438, Y  +749.026, Z    +0.000, E1   -61.150, E3 +179182.301}
SPL {X  -145.760, Y  +754.202, Z    +0.000, E1   -61.108, E3 +179187.717}
SPL {X  -143.078, Y  +758.979, Z    +0.000, E1   -60.553, E3 +179195.376}
SPL {X  -139.815, Y  +764.336, Z    +0.000, E1   -60.025, E3 +179203.228}
SPL {X  -130.672, Y  +777.307, Z    +0.000, E1   -63.098, E3 +179201.519}
SPL {X   -84.123, Y  +818.200, Z    +0.000, E1   -55.499, E3 +179315.032}
ENDSPLINE

SPLINE
SPL {X  -127.502, Y  +781.251, Z    +0.000, E1   -49.821, E3 +179447.165}
SPL {X  -151.617, Y  +742.224, Z    +0.000, E1   -39.442, E3 +179463.748}
SPL {X  -159.277, Y  +721.007, Z    +0.000, E1   -30.118, E3 +179462.925}
SPL {X  -163.701, Y  +700.836, Z    +0.000, E1   -18.960, E3 +179459.640}
SPL {X  -165.229, Y  +687.300, Z    +0.000, E1   -10.302, E3 +179459.595}
SPL {X  -165.592, Y  +679.896, Z    +0.000, E1    -5.071, E3 +179458.876}
SPL {X  -165.650, Y  +674.350, Z    +0.000, E1    -0.828, E3 +179458.250}
SPL {X  -165.650, Y  +672.653, Z    +0.000, E1    +0.827, E3 +179457.443}
SPL {X  -165.650, Y  +668.094, Z    +0.000, E1    +7.098, E3 +179456.812}
SPL {X  -165.650, Y  +662.291, Z    +0.000, E1   +16.729, E3 +179456.738}
SPL {X  -165.650, Y  +656.382, Z    +0.000, E1   +26.732, E3 +179456.296}
SPL {X  -165.650, Y  +648.240, Z    +0.000, E1   +42.276, E3 +179451.730}
SPL {X  -165.650, Y  +638.782, Z    +0.000, E1   +47.719, E3 +179458.940}
SPL {X  -165.650, Y  +622.329, Z    +0.000, E1   +68.753, E3 +179446.479}
SPL {X  -165.650, Y  +589.967, Z    +0.000, E1   +71.395, E3 +179459.105}
SPL {X  -165.650, Y  +573.012, Z    +0.000, E1   +68.475, E3 +179475.317}
SPL {X  -165.650, Y  +459.505, Z    +0.000, E1   +68.780, E3 +179547.041}
ENDSPLINE

SPLINE
SPL {X  -165.650, Y  +483.715, Z    +0.000, E1   +63.891, E3 +179563.336}
ENDSPLINE

SPLINE
SPL {X  -165.650, Y  +474.626, Z    +0.000, E1   +63.707, E3 +179573.864}
SPL {X  -165.650, Y  +465.190, Z    +0.000, E1   +63.660, E3 +179583.719}
SPL {X  -165.650, Y  +456.011, Z    +0.000, E1   +63.585, E3 +179593.614}
SPL {X  -165.650, Y  +444.310, Z    +0.000, E1   +63.666, E3 +179604.891}
SPL {X  -165.650, Y  +429.845, Z    +0.000, E1   +64.481, E3 +179613.124}
SPL {X  -165.552, Y  +372.799, Z    +0.000, E1   +69.633, E3 +179618.989}
SPL {X  -165.188, Y  +366.130, Z    +0.000, E1   +68.611, E3 +179633.391}
SPL {X  -164.361, Y  +357.877, Z    +0.000, E1   +67.700, E3 +179647.718}
SPL {X  -163.803, Y  +353.836, Z    +0.000, E1   +66.282, E3 +179662.739}
SPL {X  -162.254, Y  +345.129, Z    +0.000, E1   +65.301, E3 +179678.189}
SPL {X  -158.875, Y  +331.610, Z    +0.000, E1   +64.945, E3 +179693.248}
SPL {X  -154.872, Y  +319.724, Z    +0.000, E1   +64.496, E3 +179707.162}
SPL {X  -151.091, Y  +310.592, Z    +0.000, E1   +63.929, E3 +179719.102}
SPL {X  -148.836, Y  +305.783, Z    +0.000, E1   +63.120, E3 +179728.234}
SPL {X  -145.492, Y  +299.305, Z    +0.000, E1   +63.037, E3 +179734.726}
SPL {X  -142.120, Y  +293.401, Z    +0.000, E1   +62.602, E3 +179742.405}
SPL {X  -139.854, Y  +289.726, Z    +0.000, E1   +61.679, E3 +179750.311}
SPL {X  -135.997, Y  +283.923, Z    +0.000, E1   +62.034, E3 +179753.960}
SPL {X  -124.991, Y  +269.793, Z    +0.000, E1   +65.852, E3 +179748.949}
SPL {X   -80.641, Y  +233.804, Z    +0.000, E1   +55.283, E3 +179880.064}
ENDSPLINE

SPLINE
SPL {X  -132.197, Y  +278.681, Z    +0.000, E1   +49.692, E3 +180013.936}
SPL {X  -156.075, Y  +322.998, Z    +0.000, E1   +35.140, E3 +180019.017}
SPL {X  -162.799, Y  +347.901, Z    +0.000, E1   +22.644, E3 +180021.523}
SPL {X  -164.930, Y  +363.071, Z    +0.000, E1   +13.041, E3 +180019.263}
SPL {X  -165.629, Y  +375.893, Z    +0.000, E1    +3.908, E3 +180019.121}
SPL {X  -165.650, Y  +380.596, Z    +0.000, E1    -0.052, E3 +180017.803}
SPL {X  -165.650, Y  +383.460, Z    +0.000, E1    -3.790, E3 +180017.127}
SPL {X  -165.650, Y  +389.311, Z    +0.000, E1   -13.234, E3 +180016.613}
SPL {X  -165.650, Y  +395.103, Z    +0.000, E1   -23.932, E3 +180015.906}
SPL {X  -165.650, Y  +401.925, Z    +0.000, E1   -35.470, E3 +180015.173}
SPL {X  -165.650, Y  +410.900, Z    +0.000, E1   -46.977, E3 +180015.790}
SPL {X  -165.650, Y  +423.066, Z    +0.000, E1   -61.140, E3 +180011.521}
SPL {X  -165.650, Y  +461.121, Z    +0.000, E1   -74.504, E3 +180012.870}
SPL {X  -165.650, Y  +487.674, Z    +0.000, E1   -70.215, E3 +180035.681}
SPL {X  -165.650, Y  +590.449, Z    +0.000, E1   -68.990, E3 +180103.626}
ENDSPLINE

SPLINE
SPL {X  -165.650, Y  +577.071, Z    +0.000, E1   -65.152, E3 +180121.949}
ENDSPLINE

SPLINE
SPL {X  -165.650, Y  +580.077, Z    +0.000, E1   -64.018, E3 +180133.527}
SPL {X  -165.650, Y  +590.532, Z    +0.000, E1   -63.993, E3 +180144.093}
SPL {X  -165.650, Y  +600.616, Z    +0.000, E1   -64.059, E3 +180153.666}
SPL {X  -165.650, Y  +609.299, Z    +0.000, E1   -64.001, E3 +180162.691}
SPL {X  -165.650, Y  +618.778, Z    +0.000, E1   -63.957, E3 +180172.548}
SPL {X  -165.650, Y  +634.916, Z    +0.000, E1   -64.117, E3 +180187.597}
SPL {X  -165.650, Y  +648.710, Z    +0.000, E1   -63.999, E3 +180202.007}
SPL {X  -165.650, Y  +658.618, Z    +0.000, E1   -64.006, E3 +180211.825}
SPL {X  -165.650, Y  +670.604, Z    +0.000, E1   -64.021, E3 +180223.738}
SPL {X  -165.270, Y  +686.708, Z    +0.000, E1   -64.001, E3 +180240.081}
SPL {X  -163.641, Y  +701.218, Z    +0.000, E1   -63.638, E3 +180257.225}
SPL {X  -161.003, Y  +714.463, Z    +0.000, E1   -63.428, E3 +180271.896}
SPL {X  -157.854, Y  +725.721, Z    +0.000, E1   -62.989, E3 +180286.145}
SPL {X  -154.742, Y  +734.618, Z    +0.000, E1   -62.412, E3 +180298.631}
SPL {X  -150.939, Y  +743.744, Z    +0.000, E1   -61.955, E3 +180310.572}
SPL {X  -146.912, Y  +752.029, Z    +0.000, E1   -61.155, E3 +180323.327}
SPL {X  -143.078, Y  +758.979, Z    +0.000, E1   -60.553, E3 +180333.307}
SPL {X  -139.815, Y  +764.336, Z    +0.000, E1   -60.025, E3 +180341.159}
SPL {X  -133.503, Y  +773.566, Z    +0.000, E1   -62.412, E3 +180339.285}
SPL {X  -122.896, Y  +786.569, Z    +0.000, E1   -64.831, E3 +180339.446}
SPL {X   -84.123, Y  +818.200, Z    +0.000, E1   -55.499, E3 +180452.963}
ENDSPLINE

SPLINE
SPL {X  -127.502, Y  +781.251, Z    +0.000, E1   -49.821, E3 +180585.096}
SPL {X  -156.175, Y  +730.721, Z    +0.000, E1   -34.737, E3 +180601.375}
SPL {X  -163.701, Y  +700.836, Z    +0.000, E1   -18.960, E3 +180597.571}
SPL {X  -165.229, Y  +687.300, Z    +0.000, E1   -10.302, E3 +180597.526}
SPL {X  -165.635, Y  +677.721, Z    +0.000, E1    -3.517, E3 +180596.658}
SPL {X  -165.650, Y  +672.966, Z    +0.000, E1    +0.394, E3 +180595.560}
SPL {X  -165.650, Y  +668.094, Z    +0.000, E1    +7.098, E3 +180594.743}
SPL {X  -165.650, Y  +661.377, Z    +0.000, E1   +18.170, E3 +180594.683}
SPL {X  -165.650, Y  +654.692, Z    +0.000, E1   +29.740, E3 +180593.931}
SPL {X  -165.650, Y  +648.240, Z    +0.000, E1   +42.276, E3 +180589.661}
SPL {X  -165.650, Y  +638.477, Z    +0.000, E1   +48.488, E3 +180596.161}
SPL {X  -165.650, Y  +615.287, Z    +0.000, E1   +74.123, E3 +180580.693}
SPL {X  -165.650, Y  +589.967, Z    +0.000, E1   +71.395, E3 +180597.036}
SPL {X  -165.650, Y  +573.012, Z    +0.000, E1   +68.475, E3 +180613.248}
SPL {X  -165.650, Y  +459.505, Z    +0.000, E1   +68.780, E3 +180684.972}
ENDSPLINE

SPLINE
SPL {X  -165.650, Y  +483.715, Z    +0.000, E1   +63.891, E3 +180701.267}
ENDSPLINE

SPLINE
SPL {X  -165.650, Y  +474.626, Z    +0.000, E1   +63.707, E3 +180711.795}
SPL {X  -165.650, Y  +465.190, Z    +0.000, E1   +63.660, E3 +180721.650}
SPL {X  -165.650, Y  +456.011, Z    +0.000, E1   +63.585, E3 +180731.545}
SPL {X  -165.650, Y  +444.310, Z    +0.000, E1   +63.666, E3 +180742.822}
SPL {X  -165.650, Y  +429.845, Z    +0.000, E1   +64.481, E3 +180751.055}
SPL {X  -165.552, Y  +372.799, Z    +0.000, E1   +69.633, E3 +180756.920}
SPL {X  -165.188, Y  +366.130, Z    +0.000, E1   +68.611, E3 +180771.322}
SPL {X  -164.361, Y  +357.877, Z    +0.000, E1   +67.700, E3 +180785.649}
SPL {X  -164.353, Y  +357.815, Z    +0.000, E1   +66.333, E3 +180796.550}
SPL {X  -163.312, Y  +350.765, Z    +0.000, E1   +66.182, E3 +180804.024}
SPL {X  -163.046, Y  +349.241, Z    +0.000, E1   +65.245, E3 +180812.596}
SPL {X  -160.229, Y  +336.468, Z    +0.000, E1   +65.236, E3 +180824.579}
SPL {X  -157.078, Y  +325.903, Z    +0.000, E1   +64.692, E3 +180838.025}
SPL {X  -154.296, Y  +318.230, Z    +0.000, E1   +64.302, E3 +180847.582}
SPL {X  -151.091, Y  +310.592, Z    +0.000, E1   +63.929, E3 +180857.033}
SPL {X  -148.836, Y  +305.783, Z    +0.000, E1   +63.120, E3 +180866.165}
SPL {X  -145.492, Y  +299.305, Z    +0.000, E1   +63.037, E3 +180872.657}
SPL {X  -142.120, Y  +293.401, Z    +0.000, E1   +62.602, E3 +180880.336}
SPL {X  -139.854, Y  +289.726, Z    +0.000, E1   +61.679, E3 +180888.242}
SPL {X  -135.997, Y  +283.923, Z    +0.000, E1   +62.034, E3 +180891.891}
SPL {X  -124.991, Y  +269.793, Z    +0.000, E1   +65.852, E3 +180886.880}
SPL {X   -80.641, Y  +233.804, Z    +0.000, E1   +55.283, E3 +181017.995}
ENDSPLINE

SPLINE
SPL {X  -126.633, Y  +271.710, Z    +0.000, E1   +51.055, E3 +181148.461}
SPL {X  -147.744, Y  +303.590, Z    +0.000, E1   +42.717, E3 +181156.953}
SPL {X  -158.730, Y  +331.121, Z    +0.000, E1   +31.334, E3 +181156.861}
SPL {X  -163.642, Y  +352.786, Z    +0.000, E1   +19.725, E3 +181158.727}
SPL {X  -165.477, Y  +370.931, Z    +0.000, E1    +7.630, E3 +181157.316}
SPL {X  -165.650, Y  +380.325, Z    +0.000, E1    +0.301, E3 +181155.831}
SPL {X  -165.650, Y  +382.256, Z    +0.000, E1    -2.219, E3 +181155.160}
SPL {X  -165.650, Y  +385.791, Z    +0.000, E1    -7.347, E3 +181154.953}
SPL {X  -165.650, Y  +392.519, Z    +0.000, E1   -19.014, E3 +181154.083}
SPL {X  -165.650, Y  +401.925, Z    +0.000, E1   -35.470, E3 +181153.104}
SPL {X  -165.650, Y  +410.900, Z    +0.000, E1   -46.977, E3 +181153.721}
SPL {X  -165.650, Y  +423.066, Z    +0.000, E1   -61.140, E3 +181149.452}
SPL {X  -165.650, Y  +461.121, Z    +0.000, E1   -74.504, E3 +181150.801}
SPL {X  -165.650, Y  +487.674, Z    +0.000, E1   -70.215, E3 +181173.612}
SPL {X  -165.650, Y  +585.482, Z    +0.000, E1   -67.026, E3 +181252.774}
ENDSPLINE

SPLINE
SPL {X  -165.650, Y  +577.780, Z    +0.000, E1   -64.060, E3 +181268.986}
ENDSPLINE

SPLINE
SPL {X  -165.650, Y  +590.532, Z    +0.000, E1   -63.993, E3 +181282.024}
SPL {X  -165.650, Y  +600.616, Z    +0.000, E1   -64.059, E3 +181291.597}
SPL {X  -165.650, Y  +609.299, Z    +0.000, E1   -64.001, E3 +181300.622}
SPL {X  -165.650, Y  +618.778, Z    +0.000, E1   -63.957, E3 +181310.479}
SPL {X  -165.650, Y  +627.902, Z    +0.000, E1   -63.871, E3 +181320.206}
SPL {X  -165.650, Y  +640.120, Z    +0.000, E1   -64.248, E3 +181329.546}
SPL {X  -165.650, Y  +648.710, Z    +0.000, E1   -63.999, E3 +181339.938}
SPL {X  -165.650, Y  +658.618, Z    +0.000, E1   -64.006, E3 +181349.756}
SPL {X  -165.650, Y  +670.604, Z    +0.000, E1   -64.021, E3 +181361.669}
SPL {X  -165.270, Y  +686.708, Z    +0.000, E1   -64.001, E3 +181378.012}
SPL {X  -163.641, Y  +701.218, Z    +0.000, E1   -63.638, E3 +181395.156}
SPL {X  -161.003, Y  +714.463, Z    +0.000, E1   -63.428, E3 +181409.827}
SPL {X  -158.978, Y  +722.038, Z    +0.000, E1   -63.038, E3 +181419.895}
SPL {X  -157.142, Y  +727.904, Z    +0.000, E1   -62.905, E3 +181426.662}
SPL {X  -154.742, Y  +734.618, Z    +0.000, E1   -62.412, E3 +181436.562}
SPL {X  -150.939, Y  +743.744, Z    +0.000, E1   -61.955, E3 +181448.503}
SPL {X  -148.438, Y  +749.026, Z    +0.000, E1   -61.150, E3 +181458.163}
SPL {X  -145.760, Y  +754.202, Z    +0.000, E1   -61.108, E3 +181463.580}
SPL {X  -143.078, Y  +758.979, Z    +0.000, E1   -60.553, E3 +181471.238}
SPL {X  -139.815, Y  +764.336, Z    +0.000, E1   -60.025, E3 +181479.090}
SPL {X  -130.672, Y  +777.307, Z    +0.000, E1   -63.098, E3 +181477.381}
SPL {X   -84.123, Y  +818.200, Z    +0.000, E1   -55.499, E3 +181590.894}
ENDSPLINE

SPLINE
SPL {X  -127.502, Y  +781.251, Z    +0.000, E1   -49.821, E3 +181723.027}
SPL {X  -151.617, Y  +742.224, Z    +0.000, E1   -39.442, E3 +181739.610}
SPL {X  -161.699, Y  +711.462, Z    +0.000, E1   -25.093, E3 +181736.617}
SPL {X  -165.038, Y  +689.727, Z    +0.000, E1   -11.987, E3 +181735.654}
SPL {X  -165.635, Y  +677.721, Z    +0.000, E1    -3.517, E3 +181734.589}
SPL {X  -165.650, Y  +673.529, Z    +0.000, E1    -0.069, E3 +181733.716}
SPL {X  -165.650, Y  +670.816, Z    +0.000, E1    +3.131, E3 +181733.109}
SPL {X  -165.650, Y  +666.496, Z    +0.000, E1    +9.886, E3 +181732.183}
SPL {X  -165.650, Y  +661.377, Z    +0.000, E1   +18.170, E3 +181732.614}
SPL {X  -165.650, Y  +654.692, Z    +0.000, E1   +29.740, E3 +181731.863}
SPL {X  -165.650, Y  +648.240, Z    +0.000, E1   +42.276, E3 +181727.592}
SPL {X  -165.650, Y  +638.477, Z    +0.000, E1   +48.488, E3 +181734.092}
SPL {X  -165.650, Y  +615.287, Z    +0.000, E1   +74.123, E3 +181718.624}
SPL {X  -165.650, Y  +589.967, Z    +0.000, E1   +71.395, E3 +181734.967}
SPL {X  -165.650, Y  +573.012, Z    +0.000, E1   +68.475, E3 +181751.179}
SPL {X  -165.650, Y  +459.505, Z    +0.000, E1   +68.780, E3 +181822.903}
ENDSPLINE

SPLINE
SPL {X  -165.650, Y  +483.715, Z    +0.000, E1   +63.891, E3 +181839.198}
ENDSPLINE

SPLINE
SPL {X  -165.650, Y  +474.626, Z    +0.000, E1   +63.707, E3 +181849.727}
SPL {X  -165.650, Y  +465.190, Z    +0.000, E1   +63.660, E3 +181859.581}
SPL {X  -165.650, Y  +456.011, Z    +0.000, E1   +63.585, E3 +181869.476}
SPL {X  -165.650, Y  +441.325, Z    +0.000, E1   +63.847, E3 +181882.445}
SPL {X  -165.552, Y  +372.799, Z    +0.000, E1   +69.633, E3 +181894.851}
SPL {X  -165.443, Y  +370.231, Z    +0.000, E1   +68.724, E3 +181904.781}
SPL {X  -164.776, Y  +361.504, Z    +0.000, E1   +68.225, E3 +181916.256}
SPL {X  -164.241, Y  +356.944, Z    +0.000, E1   +66.930, E3 +181930.778}
SPL {X  -163.312, Y  +350.765, Z    +0.000, E1   +66.182, E3 +181941.955}
SPL {X  -163.046, Y  +349.241, Z    +0.000, E1   +65.245, E3 +181950.527}
SPL {X  -160.229, Y  +336.468, Z    +0.000, E1   +65.236, E3 +181962.510}
SPL {X  -157.078, Y  +325.903, Z    +0.000, E1   +64.692, E3 +181975.956}
SPL {X  -153.279, Y  +315.688, Z    +0.000, E1   +64.219, E3 +181988.529}
SPL {X  -149.447, Y  +307.046, Z    +0.000, E1   +63.460, E3 +182001.114}
SPL {X  -145.492, Y  +299.305, Z    +0.000, E1   +63.037, E3 +182010.588}
SPL {X  -142.120, Y  +293.401, Z    +0.000, E1   +62.602, E3 +182018.267}
SPL {X  -139.854, Y  +289.726, Z    +0.000, E1   +61.679, E3 +182026.173}
SPL {X  -135.997, Y  +283.923, Z    +0.000, E1   +62.034, E3 +182029.822}
SPL {X  -124.991, Y  +269.793, Z    +0.000, E1   +65.852, E3 +182024.811}
SPL {X   -80.641, Y  +233.804, Z    +0.000, E1   +55.283, E3 +182155.926}
ENDSPLINE

SPLINE
SPL {X  -132.197, Y  +278.681, Z    +0.000, E1   +49.692, E3 +182289.798}
SPL {X  -156.075, Y  +322.998, Z    +0.000, E1   +35.140, E3 +182294.879}
SPL {X  -162.799, Y  +347.901, Z    +0.000, E1   +22.644, E3 +182297.385}
SPL {X  -164.930, Y  +363.071, Z    +0.000, E1   +13.041, E3 +182295.125}
SPL {X  -165.629, Y  +375.893, Z    +0.000, E1    +3.908, E3 +182294.983}
SPL {X  -165.650, Y  +380.596, Z    +0.000, E1    -0.052, E3 +182293.665}
SPL {X  -165.650, Y  +383.460, Z    +0.000, E1    -3.790, E3 +182292.990}
SPL {X  -165.650, Y  +389.311, Z    +0.000, E1   -13.234, E3 +182292.475}
SPL {X  -165.650, Y  +395.103, Z    +0.000, E1   -23.932, E3 +182291.768}
SPL {X  -165.650, Y  +401.925, Z    +0.000, E1   -35.470, E3 +182291.035}
SPL {X  -165.650, Y  +410.900, Z    +0.000, E1   -46.977, E3 +182291.652}
SPL {X  -165.650, Y  +420.865, Z    +0.000, E1   -58.704, E3 +182288.543}
SPL {X  -165.650, Y  +450.181, Z    +0.000, E1   -73.218, E3 +182286.491}
SPL {X  -165.650, Y  +487.674, Z    +0.000, E1   -70.215, E3 +182311.543}
SPL {X  -165.650, Y  +590.449, Z    +0.000, E1   -68.990, E3 +182379.488}
ENDSPLINE

SPLINE
SPL {X  -165.650, Y  +577.071, Z    +0.000, E1   -65.152, E3 +182397.811}
ENDSPLINE

SPLINE
SPL {X  -165.650, Y  +580.077, Z    +0.000, E1   -64.018, E3 +182409.389}
SPL {X  -165.650, Y  +590.532, Z    +0.000, E1   -63.993, E3 +182419.955}
SPL {X  -165.650, Y  +604.471, Z    +0.000, E1   -64.071, E3 +182433.462}
SPL {X  -165.650, Y  +618.778, Z    +0.000, E1   -63.957, E3 +182448.410}
SPL {X  -165.650, Y  +634.916, Z    +0.000, E1   -64.117, E3 +182463.459}
SPL {X  -165.650, Y  +648.710, Z    +0.000, E1   -63.999, E3 +182477.869}
SPL {X  -165.650, Y  +658.618, Z    +0.000, E1   -64.006, E3 +182487.687}
SPL {X  -165.650, Y  +670.604, Z    +0.000, E1   -64.021, E3 +182499.600}
SPL {X  -165.553, Y  +681.156, Z    +0.000, E1   -63.834, E3 +182511.475}
SPL {X  -164.902, Y  +691.221, Z    +0.000, E1   -64.073, E3 +182519.734}
SPL {X  -163.641, Y  +701.218, Z    +0.000, E1   -63.638, E3 +182533.087}
SPL {X  -161.003, Y  +714.463, Z    +0.000, E1   -63.428, E3 +182547.758}
SPL {X  -158.978, Y  +722.038, Z    +0.000, E1   -63.038, E3 +182557.826}
SPL {X  -156.651, Y  +729.355, Z    +0.000, E1   -62.675, E3 +182567.741}
SPL {X  -153.281, Y  +738.308, Z    +0.000, E1   -62.233, E3 +182579.341}
SPL {X  -150.070, Y  +745.636, Z    +0.000, E1   -61.982, E3 +182588.088}
SPL {X  -146.912, Y  +752.029, Z    +0.000, E1   -61.155, E3 +182599.190}
SPL {X  -143.078, Y  +758.979, Z    +0.000, E1   -60.553, E3 +182609.169}
SPL {X  -139.815, Y  +764.336, Z    +0.000, E1   -60.025, E3 +182617.021}
SPL {X  -130.672, Y  +777.307, Z    +0.000, E1   -63.098, E3 +182615.312}
SPL {X   -84.123, Y  +818.200, Z    +0.000, E1   -55.499, E3 +182728.825}
ENDSPLINE

SPLINE
SPL {X  -127.502, Y  +781.251, Z    +0.000, E1   -49.821, E3 +182860.958}
SPL {X  -156.175, Y  +730.721, Z    +0.000, E1   -34.737, E3 +182877.238}
SPL {X  -163.701, Y  +700.836, Z    +0.000, E1   -18.960, E3 +182873.433}
SPL {X  -165.229, Y  +687.300, Z    +0.000, E1   -10.302, E3 +182873.388}
SPL {X  -165.635, Y  +677.721, Z    +0.000, E1    -3.517, E3 +182872.520}
SPL {X  -165.650, Y  +672.966, Z    +0.000, E1    +0.394, E3 +182871.423}
SPL {X  -165.650, Y  +668.094, Z    +0.000, E1    +7.098, E3 +182870.606}
SPL {X  -165.650, Y  +662.291, Z    +0.000, E1   +16.729, E3 +182870.531}
SPL {X  -165.650, Y  +656.382, Z    +0.000, E1   +26.732, E3 +182870.089}
SPL {X  -165.650, Y  +648.240, Z    +0.000, E1   +42.276, E3 +182865.523}
SPL {X  -165.650, Y  +638.477, Z    +0.000, E1   +48.488, E3 +182872.023}
SPL {X  -165.650, Y  +615.287, Z    +0.000, E1   +74.123, E3 +182856.555}
SPL {X  -165.650, Y  +589.967, Z    +0.000, E1   +71.395, E3 +182872.898}
SPL {X  -165.650, Y  +573.012, Z    +0.000, E1   +68.475, E3 +182889.110}
SPL {X  -165.650, Y  +459.505, Z    +0.000, E1   +68.780, E3 +182960.834}
ENDSPLINE

SPLINE
SPL {X  -165.650, Y  +483.715, Z    +0.000, E1   +63.891, E3 +182977.129}
ENDSPLINE

SPLINE
SPL {X  -165.650, Y  +474.626, Z    +0.000, E1   +63.707, E3 +182987.658}
SPL {X  -165.650, Y  +465.190, Z    +0.000, E1   +63.660, E3 +182997.512}
SPL {X  -165.650, Y  +456.011, Z    +0.000, E1   +63.585, E3 +183007.407}
SPL {X  -165.650, Y  +441.325, Z    +0.000, E1   +63.847, E3 +183020.376}
SPL {X  -165.552, Y  +372.799, Z    +0.000, E1   +69.633, E3 +183032.782}
SPL {X  -165.188, Y  +366.130, Z    +0.000, E1   +68.611, E3 +183047.184}
SPL {X  -164.361, Y  +357.877, Z    +0.000, E1   +67.700, E3 +183061.511}
SPL {X  -164.353, Y  +357.815, Z    +0.000, E1   +66.333, E3 +183072.412}
SPL {X  -163.312, Y  +350.765, Z    +0.000, E1   +66.182, E3 +183079.886}
SPL {X  -163.046, Y  +349.241, Z    +0.000, E1   +65.245, E3 +183088.458}
SPL {X  -160.229, Y  +336.468, Z    +0.000, E1   +65.236, E3 +183100.441}
SPL {X  -158.158, Y  +329.247, Z    +0.000, E1   +64.622, E3 +183111.213}
SPL {X  -154.872, Y  +319.724, Z    +0.000, E1   +64.496, E3 +183120.955}
SPL {X  -151.091, Y  +310.592, Z    +0.000, E1   +63.929, E3 +183132.895}
SPL {X  -148.836, Y  +305.783, Z    +0.000, E1   +63.120, E3 +183142.027}
SPL {X  -145.492, Y  +299.305, Z    +0.000, E1   +63.037, E3 +183148.519}
SPL {X  -142.120, Y  +293.401, Z    +0.000, E1   +62.602, E3 +183156.198}
SPL {X  -139.854, Y  +289.726, Z    +0.000, E1   +61.679, E3 +183164.104}
SPL {X  -135.997, Y  +283.923, Z    +0.000, E1   +62.034, E3 +183167.753}
SPL {X  -124.991, Y  +269.793, Z    +0.000, E1   +65.852, E3 +183162.742}
SPL {X   -80.641, Y  +233.804, Z    +0.000, E1   +55.283, E3 +183293.857}
ENDSPLINE

SPLINE
SPL {X  -132.197, Y  +278.681, Z    +0.000, E1   +49.692, E3 +183427.729}
SPL {X  -156.075, Y  +322.998, Z    +0.000, E1   +35.140, E3 +183432.810}
SPL {X  -163.642, Y  +352.786, Z    +0.000, E1   +19.725, E3 +183434.589}
SPL {X  -165.477, Y  +370.931, Z    +0.000, E1    +7.630, E3 +183433.178}
SPL {X  -165.650, Y  +378.219, Z    +0.000, E1    +1.951, E3 +183432.451}
SPL {X  -165.650, Y  +380.596, Z    +0.000, E1    -0.052, E3 +183431.596}
SPL {X  -165.650, Y  +383.460, Z    +0.000, E1    -3.790, E3 +183430.921}
SPL {X  -165.650, Y  +387.326, Z    +0.000, E1   -10.041, E3 +183430.792}
SPL {X  -165.650, Y  +392.519, Z    +0.000, E1   -19.014, E3 +183429.945}
SPL {X  -165.650, Y  +401.925, Z    +0.000, E1   -35.470, E3 +183428.966}
SPL {X  -165.650, Y  +410.900, Z    +0.000, E1   -46.977, E3 +183429.583}
SPL {X  -165.650, Y  +420.865, Z    +0.000, E1   -58.704, E3 +183426.474}
SPL {X  -165.650, Y  +450.181, Z    +0.000, E1   -73.218, E3 +183424.422}
SPL {X  -165.650, Y  +487.674, Z    +0.000, E1   -70.215, E3 +183449.474}
SPL {X  -165.650, Y  +585.482, Z    +0.000, E1   -67.026, E3 +183528.636}
ENDSPLINE

SPLINE
SPL {X  -165.650, Y  +571.836, Z    +0.000, E1   -64.066, E3 +183538.657}
ENDSPLINE

SPLINE
SPL {X  -165.650, Y  +580.077, Z    +0.000, E1   -64.018, E3 +183547.320}
SPL {X  -165.650, Y  +590.532, Z    +0.000, E1   -63.993, E3 +183557.886}
SPL {X  -165.650, Y  +604.471, Z    +0.000, E1   -64.071, E3 +183571.393}
SPL {X  -165.650, Y  +618.778, Z    +0.000, E1   -63.957, E3 +183586.341}
SPL {X  -165.650, Y  +627.902, Z    +0.000, E1   -63.871, E3 +183596.068}
SPL {X  -165.650, Y  +640.120, Z    +0.000, E1   -64.248, E3 +183605.409}
SPL {X  -165.650, Y  +648.710, Z    +0.000, E1   -63.999, E3 +183615.801}
SPL {X  -165.650, Y  +658.618, Z    +0.000, E1   -64.006, E3 +183625.618}
SPL {X  -165.650, Y  +670.604, Z    +0.000, E1   -64.021, E3 +183637.531}
SPL {X  -165.270, Y  +686.708, Z    +0.000, E1   -64.001, E3 +183653.874}
SPL {X  -163.641, Y  +701.218, Z    +0.000, E1   -63.638, E3 +183671.018}
SPL {X  -161.003, Y  +714.463, Z    +0.000, E1   -63.428, E3 +183685.689}
SPL {X  -157.854, Y  +725.721, Z    +0.000, E1   -62.989, E3 +183699.938}
SPL {X  -154.742, Y  +734.618, Z    +0.000, E1   -62.412, E3 +183712.424}
SPL {X  -150.939, Y  +743.744, Z    +0.000, E1   -61.955, E3 +183724.365}
SPL {X  -146.912, Y  +752.029, Z    +0.000, E1   -61.155, E3 +183737.121}
SPL {X  -143.078, Y  +758.979, Z    +0.000, E1   -60.553, E3 +183747.100}
SPL {X  -139.815, Y  +764.336, Z    +0.000, E1   -60.025, E3 +183754.952}
SPL {X  -130.672, Y  +777.307, Z    +0.000, E1   -63.098, E3 +183753.243}
SPL {X   -84.123, Y  +818.200, Z    +0.000, E1   -55.499, E3 +183866.756}
ENDSPLINE

SPLINE
SPL {X  -127.502, Y  +781.251, Z    +0.000, E1   -49.821, E3 +183998.889}
SPL {X  -151.617, Y  +742.224, Z    +0.000, E1   -39.442, E3 +184015.472}
SPL {X  -159.277, Y  +721.007, Z    +0.000, E1   -30.118, E3 +184014.649}
SPL {X  -163.701, Y  +700.836, Z    +0.000, E1   -18.960, E3 +184011.364}
SPL {X  -165.229, Y  +687.300, Z    +0.000, E1   -10.302, E3 +184011.319}
SPL {X  -165.592, Y  +679.896, Z    +0.000, E1    -5.071, E3 +184010.600}
SPL {X  -165.650, Y  +673.846, Z    +0.000, E1    -0.441, E3 +184009.680}
SPL {X  -165.650, Y  +670.816, Z    +0.000, E1    +3.131, E3 +184008.971}
SPL {X  -165.650, Y  +666.496, Z    +0.000, E1    +9.886, E3 +184008.045}
SPL {X  -165.650, Y  +661.377, Z    +0.000, E1   +18.170, E3 +184008.476}
SPL {X  -165.650, Y  +654.692, Z    +0.000, E1   +29.740, E3 +184007.725}
SPL {X  -165.650, Y  +648.240, Z    +0.000, E1   +42.276, E3 +184003.454}
SPL {X  -165.650, Y  +638.477, Z    +0.000, E1   +48.488, E3 +184009.954}
SPL {X  -165.650, Y  +615.287, Z    +0.000, E1   +74.123, E3 +183994.486}
SPL {X  -165.650, Y  +589.967, Z    +0.000, E1   +71.395, E3 +184010.829}
SPL {X  -165.650, Y  +573.012, Z    +0.000, E1   +68.475, E3 +184027.042}
SPL {X  -165.650, Y  +459.505, Z    +0.000, E1   +68.780, E3 +184098.765}
ENDSPLINE

SPLINE
SPL {X  -165.650, Y  +483.715, Z    +0.000, E1   +63.891, E3 +184115.060}
ENDSPLINE

SPLINE
SPL {X  -165.650, Y  +474.626, Z    +0.000, E1   +63.707, E3 +184125.589}
SPL {X  -165.650, Y  +465.190, Z    +0.000, E1   +63.660, E3 +184135.443}
SPL {X  -165.650, Y  +456.011, Z    +0.000, E1   +63.585, E3 +184145.338}
SPL {X  -165.650, Y  +441.325, Z    +0.000, E1   +63.847, E3 +184158.307}
SPL {X  -165.552, Y  +372.799, Z    +0.000, E1   +69.633, E3 +184170.713}
SPL {X  -165.443, Y  +370.231, Z    +0.000, E1   +68.724, E3 +184180.643}
SPL {X  -164.776, Y  +361.504, Z    +0.000, E1   +68.225, E3 +184192.118}
SPL {X  -164.137, Y  +356.163, Z    +0.000, E1   +67.495, E3 +184202.408}
SPL {X  -163.803, Y  +353.836, Z    +0.000, E1   +66.282, E3 +184214.463}
SPL {X  -162.254, Y  +345.129, Z    +0.000, E1   +65.301, E3 +184229.914}
SPL {X  -158.875, Y  +331.610, Z    +0.000, E1   +64.945, E3 +184244.972}
SPL {X  -154.872, Y  +319.724, Z    +0.000, E1   +64.496, E3 +184258.886}
SPL {X  -151.091, Y  +310.592, Z    +0.000, E1   +63.929, E3 +184270.826}
SPL {X  -148.836, Y  +305.783, Z    +0.000, E1   +63.120, E3 +184279.958}
SPL {X  -145.492, Y  +299.305, Z    +0.000, E1   +63.037, E3 +184286.450}
SPL {X  -142.120, Y  +293.401, Z    +0.000, E1   +62.602, E3 +184294.129}
SPL {X  -139.854, Y  +289.726, Z    +0.000, E1   +61.679, E3 +184302.035}
SPL {X  -135.997, Y  +283.923, Z    +0.000, E1   +62.034, E3 +184305.684}
SPL {X  -124.991, Y  +269.793, Z    +0.000, E1   +65.852, E3 +184300.673}
SPL {X   -80.641, Y  +233.804, Z    +0.000, E1   +55.283, E3 +184431.788}
ENDSPLINE

SPLINE
SPL {X  -126.633, Y  +271.710, Z    +0.000, E1   +51.055, E3 +184562.254}
SPL {X  -147.744, Y  +303.590, Z    +0.000, E1   +42.717, E3 +184570.746}
SPL {X  -158.730, Y  +331.121, Z    +0.000, E1   +31.334, E3 +184570.654}
SPL {X  -162.799, Y  +347.901, Z    +0.000, E1   +22.644, E3 +184573.247}
SPL {X  -164.930, Y  +363.071, Z    +0.000, E1   +13.041, E3 +184570.987}
SPL {X  -165.629, Y  +375.893, Z    +0.000, E1    +3.908, E3 +184570.845}
SPL {X  -165.650, Y  +380.596, Z    +0.000, E1    -0.052, E3 +184569.527}
SPL {X  -165.650, Y  +382.256, Z    +0.000, E1    -2.219, E3 +184568.954}
SPL {X  -165.650, Y  +385.791, Z    +0.000, E1    -7.347, E3 +184568.746}
SPL {X  -165.650, Y  +392.519, Z    +0.000, E1   -19.014, E3 +184567.876}
SPL {X  -165.650, Y  +401.925, Z    +0.000, E1   -35.470, E3 +184566.897}
SPL {X  -165.650, Y  +410.900, Z    +0.000, E1   -46.977, E3 +184567.514}
SPL {X  -165.650, Y  +420.865, Z    +0.000, E1   -58.704, E3 +184564.405}
SPL {X  -165.650, Y  +450.181, Z    +0.000, E1   -73.218, E3 +184562.353}
SPL {X  -165.650, Y  +487.674, Z    +0.000, E1   -70.215, E3 +184587.405}
SPL {X  -165.650, Y  +590.449, Z    +0.000, E1   -68.990, E3 +184655.350}
ENDSPLINE

SPLINE
SPL {X  -165.650, Y  +577.071, Z    +0.000, E1   -65.152, E3 +184673.673}
ENDSPLINE

SPLINE
SPL {X  -165.650, Y  +580.077, Z    +0.000, E1   -64.018, E3 +184685.251}
SPL {X  -165.650, Y  +590.532, Z    +0.000, E1   -63.993, E3 +184695.817}
SPL {X  -165.650, Y  +604.471, Z    +0.000, E1   -64.071, E3 +184709.325}
SPL {X  -165.650, Y  +618.778, Z    +0.000, E1   -63.957, E3 +184724.272}
SPL {X  -165.650, Y  +634.916, Z    +0.000, E1   -64.117, E3 +184739.321}
SPL {X  -165.650, Y  +648.710, Z    +0.000, E1   -63.999, E3 +184753.732}
SPL {X  -165.650, Y  +660.990, Z    +0.000, E1   -63.976, E3 +184766.257}
SPL {X  -165.633, Y  +677.852, Z    +0.000, E1   -63.999, E3 +184783.030}
SPL {X  -164.651, Y  +693.668, Z    +0.000, E1   -63.860, E3 +184799.862}
SPL {X  -163.017, Y  +704.915, Z    +0.000, E1   -63.665, E3 +184812.305}
SPL {X  -161.003, Y  +714.463, Z    +0.000, E1   -63.428, E3 +184823.620}
SPL {X  -157.854, Y  +725.721, Z    +0.000, E1   -62.989, E3 +184837.869}
SPL {X  -155.984, Y  +731.258, Z    +0.000, E1   -62.241, E3 +184848.015}
SPL {X  -153.281, Y  +738.308, Z    +0.000, E1   -62.233, E3 +184855.203}
SPL {X  -150.070, Y  +745.636, Z    +0.000, E1   -61.982, E3 +184863.950}
SPL {X  -148.438, Y  +749.026, Z    +0.000, E1   -61.150, E3 +184871.956}
SPL {X  -145.760, Y  +754.202, Z    +0.000, E1   -61.108, E3 +184877.373}
SPL {X  -143.078, Y  +758.979, Z    +0.000, E1   -60.553, E3 +184885.031}
SPL {X  -139.815, Y  +764.336, Z    +0.000, E1   -60.025, E3 +184892.883}
SPL {X  -130.672, Y  +777.307, Z    +0.000, E1   -63.098, E3 +184891.174}
SPL {X   -84.123, Y  +818.200, Z    +0.000, E1   -55.499, E3 +185004.687}
ENDSPLINE

SPLINE
SPL {X  -127.502, Y  +781.251, Z    +0.000, E1   -49.821, E3 +185136.820}
SPL {X  -151.617, Y  +742.224, Z    +0.000, E1   -39.442, E3 +185153.403}
SPL {X  -159.277, Y  +721.007, Z    +0.000, E1   -30.118, E3 +185152.580}
SPL {X  -163.701, Y  +700.836, Z    +0.000, E1   -18.960, E3 +185149.295}
SPL {X  -165.229, Y  +687.300, Z    +0.000, E1   -10.302, E3 +185149.250}
SPL {X  -165.592, Y  +679.896, Z    +0.000, E1    -5.071, E3 +185148.531}
SPL {X  -165.650, Y  +673.846, Z    +0.000, E1    -0.441, E3 +185147.611}
SPL {X  -165.650, Y  +670.816, Z    +0.000, E1    +3.131, E3 +185146.902}
SPL {X  -165.650, Y  +666.496, Z    +0.000, E1    +9.886, E3 +185145.976}
SPL {X  -165.650, Y  +661.377, Z    +0.000, E1   +18.170, E3 +185146.407}
SPL {X  -165.650, Y  +654.692, Z    +0.000, E1   +29.740, E3 +185145.656}
SPL {X  -165.650, Y  +648.240, Z    +0.000, E1   +42.276, E3 +185141.385}
SPL {X  -165.650, Y  +638.477, Z    +0.000, E1   +48.488, E3 +185147.886}
SPL {X  -165.650, Y  +615.287, Z    +0.000, E1   +74.123, E3 +185132.417}
SPL {X  -165.650, Y  +589.967, Z    +0.000, E1   +71.395, E3 +185148.760}
SPL {X  -165.650, Y  +573.012, Z    +0.000, E1   +68.475, E3 +185164.973}
SPL {X  -165.650, Y  +459.505, Z    +0.000, E1   +68.780, E3 +185236.696}
ENDSPLINE

SPLINE
SPL {X  -165.650, Y  +483.715, Z    +0.000, E1   +63.891, E3 +185252.991}
ENDSPLINE

SPLINE
SPL {X  -165.650, Y  +474.626, Z    +0.000, E1   +63.707, E3 +185263.520}
SPL {X  -165.650, Y  +465.190, Z    +0.000, E1   +63.660, E3 +185273.374}
SPL {X  -165.650, Y  +456.011, Z    +0.000, E1   +63.585, E3 +185283.269}
SPL {X  -165.650, Y  +444.310, Z    +0.000, E1   +63.666, E3 +185294.546}
SPL {X  -165.650, Y  +429.845, Z    +0.000, E1   +64.481, E3 +185302.779}
SPL {X  -165.552, Y  +372.799, Z    +0.000, E1   +69.633, E3 +185308.644}
SPL {X  -165.188, Y  +366.130, Z    +0.000, E1   +68.611, E3 +185323.046}
SPL {X  -164.361, Y  +357.877, Z    +0.000, E1   +67.700, E3 +185337.373}
SPL {X  -164.353, Y  +357.815, Z    +0.000, E1   +66.333, E3 +185348.275}
SPL {X  -163.312, Y  +350.765, Z    +0.000, E1   +66.182, E3 +185355.748}
SPL {X  -163.046, Y  +349.241, Z    +0.000, E1   +65.245, E3 +185364.320}
SPL {X  -160.229, Y  +336.468, Z    +0.000, E1   +65.236, E3 +185376.303}
SPL {X  -158.158, Y  +329.247, Z    +0.000, E1   +64.622, E3 +185387.075}
SPL {X  -154.872, Y  +319.724, Z    +0.000, E1   +64.496, E3 +185396.817}
SPL {X  -151.091, Y  +310.592, Z    +0.000, E1   +63.929, E3 +185408.757}
SPL {X  -148.836, Y  +305.783, Z    +0.000, E1   +63.120, E3 +185417.889}
SPL {X  -145.492, Y  +299.305, Z    +0.000, E1   +63.037, E3 +185424.381}
SPL {X  -142.120, Y  +293.401, Z    +0.000, E1   +62.602, E3 +185432.060}
SPL {X  -139.854, Y  +289.726, Z    +0.000, E1   +61.679, E3 +185439.966}
SPL {X  -135.997, Y  +283.923, Z    +0.000, E1   +62.034, E3 +185443.615}
SPL {X  -124.991, Y  +269.793, Z    +0.000, E1   +65.852, E3 +185438.604}
SPL {X   -80.641, Y  +233.804, Z    +0.000, E1   +55.283, E3 +185569.719}
ENDSPLINE

SPLINE
SPL {X  -132.197, Y  +278.681, Z    +0.000, E1   +49.692, E3 +185703.592}
SPL {X  -156.075, Y  +322.998, Z    +0.000, E1   +35.140, E3 +185708.672}
SPL {X  -163.642, Y  +352.786, Z    +0.000, E1   +19.725, E3 +185710.451}
SPL {X  -165.477, Y  +370.931, Z    +0.000, E1    +7.630, E3 +185709.040}
SPL {X  -165.650, Y  +378.219, Z    +0.000, E1    +1.951, E3 +185708.313}
SPL {X  -165.650, Y  +381.007, Z    +0.000, E1    -0.398, E3 +185707.316}
SPL {X  -165.650, Y  +385.791, Z    +0.000, E1    -7.347, E3 +185706.677}
SPL {X  -165.650, Y  +390.879, Z    +0.000, E1   -16.263, E3 +185705.963}
SPL {X  -165.650, Y  +395.103, Z    +0.000, E1   -23.932, E3 +185705.561}
SPL {X  -165.650, Y  +401.925, Z    +0.000, E1   -35.470, E3 +185704.828}
SPL {X  -165.650, Y  +410.900, Z    +0.000, E1   -46.977, E3 +185705.445}
SPL {X  -165.650, Y  +423.066, Z    +0.000, E1   -61.140, E3 +185701.176}
SPL {X  -165.650, Y  +461.121, Z    +0.000, E1   -74.504, E3 +185702.525}
SPL {X  -165.650, Y  +487.674, Z    +0.000, E1   -70.215, E3 +185725.336}
SPL {X  -165.650, Y  +585.482, Z    +0.000, E1   -67.026, E3 +185804.498}
ENDSPLINE

SPLINE
SPL {X  -165.650, Y  +577.780, Z    +0.000, E1   -64.060, E3 +185820.710}
ENDSPLINE

SPLINE
SPL {X  -165.650, Y  +590.532, Z    +0.000, E1   -63.993, E3 +185833.748}
SPL {X  -165.650, Y  +600.616, Z    +0.000, E1   -64.059, E3 +185843.322}
SPL {X  -165.650, Y  +609.299, Z    +0.000, E1   -64.001, E3 +185852.347}
SPL {X  -165.650, Y  +618.778, Z    +0.000, E1   -63.957, E3 +185862.204}
SPL {X  -165.650, Y  +627.902, Z    +0.000, E1   -63.871, E3 +185871.930}
SPL {X  -165.650, Y  +640.120, Z    +0.000, E1   -64.248, E3 +185881.271}
SPL {X  -165.650, Y  +648.710, Z    +0.000, E1   -63.999, E3 +185891.663}
SPL {X  -165.650, Y  +658.618, Z    +0.000, E1   -64.006, E3 +185901.480}
SPL {X  -165.650, Y  +670.604, Z    +0.000, E1   -64.021, E3 +185913.393}
SPL {X  -165.270, Y  +686.708, Z    +0.000, E1   -64.001, E3 +185929.736}
SPL {X  -163.641, Y  +701.218, Z    +0.000, E1   -63.638, E3 +185946.880}
SPL {X  -161.003, Y  +714.463, Z    +0.000, E1   -63.428, E3 +185961.551}
SPL {X  -158.978, Y  +722.038, Z    +0.000, E1   -63.038, E3 +185971.619}
SPL {X  -156.651, Y  +729.355, Z    +0.000, E1   -62.675, E3 +185981.534}
SPL {X  -153.281, Y  +738.308, Z    +0.000, E1   -62.233, E3 +185993.134}
SPL {X  -150.070, Y  +745.636, Z    +0.000, E1   -61.982, E3 +186001.881}
SPL {X  -146.912, Y  +752.029, Z    +0.000, E1   -61.155, E3 +186012.983}
SPL {X  -143.078, Y  +758.979, Z    +0.000, E1   -60.553, E3 +186022.962}
SPL {X  -139.815, Y  +764.336, Z    +0.000, E1   -60.025, E3 +186030.814}
SPL {X  -130.672, Y  +777.307, Z    +0.000, E1   -63.098, E3 +186029.105}
SPL {X   -84.123, Y  +818.200, Z    +0.000, E1   -55.499, E3 +186142.618}
ENDSPLINE

SPLINE
SPL {X  -116.242, Y  +793.515, Z    +0.000, E1   -51.439, E3 +186260.491}
SPL {X  -136.975, Y  +768.655, Z    +0.000, E1   -47.464, E3 +186284.947}
SPL {X  -151.617, Y  +742.224, Z    +0.000, E1   -39.442, E3 +186291.334}
SPL {X  -161.699, Y  +711.462, Z    +0.000, E1   -25.093, E3 +186288.341}
SPL {X  -165.038, Y  +689.727, Z    +0.000, E1   -11.987, E3 +186287.378}
SPL {X  -165.592, Y  +679.896, Z    +0.000, E1    -5.071, E3 +186286.462}
SPL {X  -165.650, Y  +674.350, Z    +0.000, E1    -0.828, E3 +186285.836}
SPL {X  -165.650, Y  +672.653, Z    +0.000, E1    +0.827, E3 +186285.029}
SPL {X  -165.650, Y  +669.589, Z    +0.000, E1    +5.031, E3 +186284.858}
SPL {X  -165.650, Y  +666.496, Z    +0.000, E1    +9.886, E3 +186283.907}
SPL {X  -165.650, Y  +662.291, Z    +0.000, E1   +16.729, E3 +186284.324}
SPL {X  -165.650, Y  +656.382, Z    +0.000, E1   +26.732, E3 +186283.882}
SPL {X  -165.650, Y  +648.240, Z    +0.000, E1   +42.276, E3 +186279.316}
SPL {X  -165.650, Y  +638.477, Z    +0.000, E1   +48.488, E3 +186285.817}
SPL {X  -165.650, Y  +615.287, Z    +0.000, E1   +74.123, E3 +186270.348}
SPL {X  -165.650, Y  +589.967, Z    +0.000, E1   +71.395, E3 +186286.691}
SPL {X  -165.650, Y  +573.012, Z    +0.000, E1   +68.475, E3 +186302.904}
SPL {X  -165.650, Y  +459.505, Z    +0.000, E1   +68.780, E3 +186374.627}
ENDSPLINE

SPLINE
SPL {X  -165.650, Y  +483.715, Z    +0.000, E1   +63.891, E3 +186390.922}
ENDSPLINE

SPLINE
SPL {X  -165.650, Y  +474.626, Z    +0.000, E1   +63.707, E3 +186401.451}
SPL {X  -165.650, Y  +465.190, Z    +0.000, E1   +63.660, E3 +186411.305}
SPL {X  -165.650, Y  +456.011, Z    +0.000, E1   +63.585, E3 +186421.200}
SPL {X  -165.650, Y  +441.325, Z    +0.000, E1   +63.847, E3 +186434.169}
SPL {X  -165.552, Y  +372.799, Z    +0.000, E1   +69.633, E3 +186446.575}
SPL {X  -165.188, Y  +366.130, Z    +0.000, E1   +68.611, E3 +186460.977}
SPL {X  -164.361, Y  +357.877, Z    +0.000, E1   +67.700, E3 +186475.304}
SPL {X  -163.803, Y  +353.836, Z    +0.000, E1   +66.282, E3 +186490.326}
SPL {X  -162.254, Y  +345.129, Z    +0.000, E1   +65.301, E3 +186505.776}
SPL {X  -159.503, Y  +333.793, Z    +0.000, E1   +65.139, E3 +186517.220}
SPL {X  -157.078, Y  +325.903, Z    +0.000, E1   +64.692, E3 +186527.680}
SPL {X  -153.279, Y  +315.688, Z    +0.000, E1   +64.219, E3 +186540.253}
SPL {X  -149.447, Y  +307.046, Z    +0.000, E1   +63.460, E3 +186552.838}
SPL {X  -145.492, Y  +299.305, Z    +0.000, E1   +63.037, E3 +186562.312}
SPL {X  -142.120, Y  +293.401, Z    +0.000, E1   +62.602, E3 +186569.991}
SPL {X  -139.854, Y  +289.726, Z    +0.000, E1   +61.679, E3 +186577.897}
SPL {X  -135.997, Y  +283.923, Z    +0.000, E1   +62.034, E3 +186581.546}
SPL {X  -124.991, Y  +269.793, Z    +0.000, E1   +65.852, E3 +186576.535}
SPL {X   -80.641, Y  +233.804, Z    +0.000, E1   +55.283, E3 +186707.650}
ENDSPLINE

SPLINE
SPL {X  -132.197, Y  +278.681, Z    +0.000, E1   +49.692, E3 +186841.523}
SPL {X  -156.075, Y  +322.998, Z    +0.000, E1   +35.140, E3 +186846.603}
SPL {X  -163.642, Y  +352.786, Z    +0.000, E1   +19.725, E3 +186848.383}
SPL {X  -165.477, Y  +370.931, Z    +0.000, E1    +7.630, E3 +186846.971}
SPL {X  -165.650, Y  +378.219, Z    +0.000, E1    +1.951, E3 +186846.244}
SPL {X  -165.650, Y  +380.596, Z    +0.000, E1    -0.052, E3 +186845.389}
SPL {X  -165.650, Y  +383.460, Z    +0.000, E1    -3.790, E3 +186844.714}
SPL {X  -165.650, Y  +387.326, Z    +0.000, E1   -10.041, E3 +186844.585}
SPL {X  -165.650, Y  +392.519, Z    +0.000, E1   -19.014, E3 +186843.738}
SPL {X  -165.650, Y  +401.925, Z    +0.000, E1   -35.470, E3 +186842.759}
SPL {X  -165.650, Y  +410.900, Z    +0.000, E1   -46.977, E3 +186843.376}
SPL {X  -165.650, Y  +420.865, Z    +0.000, E1   -58.704, E3 +186840.267}
SPL {X  -165.650, Y  +450.181, Z    +0.000, E1   -73.218, E3 +186838.215}
SPL {X  -165.650, Y  +487.674, Z    +0.000, E1   -70.215, E3 +186863.267}
SPL {X  -165.650, Y  +585.482, Z    +0.000, E1   -67.026, E3 +186942.429}
ENDSPLINE

SPLINE
SPL {X  -165.650, Y  +577.780, Z    +0.000, E1   -64.060, E3 +186958.641}
ENDSPLINE

SPLINE
SPL {X  -165.650, Y  +590.532, Z    +0.000, E1   -63.993, E3 +186971.679}
SPL {X  -165.650, Y  +600.616, Z    +0.000, E1   -64.059, E3 +186981.253}
SPL {X  -165.650, Y  +609.299, Z    +0.000, E1   -64.001, E3 +186990.278}
SPL {X  -165.650, Y  +618.778, Z    +0.000, E1   -63.957, E3 +187000.135}
SPL {X  -165.650, Y  +634.916, Z    +0.000, E1   -64.117, E3 +187015.183}
SPL {X  -165.650, Y  +648.710, Z    +0.000, E1   -63.999, E3 +187029.594}
SPL {X  -165.650, Y  +658.618, Z    +0.000, E1   -64.006, E3 +187039.411}
SPL {X  -165.650, Y  +670.604, Z    +0.000, E1   -64.021, E3 +187051.324}
SPL {X  -165.553, Y  +681.156, Z    +0.000, E1   -63.834, E3 +187063.199}
SPL {X  -164.651, Y  +693.668, Z    +0.000, E1   -63.860, E3 +187075.724}
SPL {X  -163.017, Y  +704.915, Z    +0.000, E1   -63.665, E3 +187088.167}
SPL {X  -161.003, Y  +714.463, Z    +0.000, E1   -63.428, E3 +187099.482}
SPL {X  -157.854, Y  +725.721, Z    +0.000, E1   -62.989, E3 +187113.731}
SPL {X  -155.984, Y  +731.258, Z    +0.000, E1   -62.241, E3 +187123.877}
SPL {X  -153.281, Y  +738.308, Z    +0.000, E1   -62.233, E3 +187131.065}
SPL {X  -150.070, Y  +745.636, Z    +0.000, E1   -61.982, E3 +187139.812}
SPL {X  -146.912, Y  +752.029, Z    +0.000, E1   -61.155, E3 +187150.914}
SPL {X  -143.078, Y  +758.979, Z    +0.000, E1   -60.553, E3 +187160.893}
SPL {X  -139.815, Y  +764.336, Z    +0.000, E1   -60.025, E3 +187168.745}
SPL {X  -130.672, Y  +777.307, Z    +0.000, E1   -63.098, E3 +187167.036}
SPL {X   -84.123, Y  +818.200, Z    +0.000, E1   -55.499, E3 +187280.549}
ENDSPLINE

SPLINE
SPL {X  -127.502, Y  +781.251, Z    +0.000, E1   -49.821, E3 +187412.683}
SPL {X  -151.617, Y  +742.224, Z    +0.000, E1   -39.442, E3 +187429.265}
SPL {X  -161.699, Y  +711.462, Z    +0.000, E1   -25.093, E3 +187426.272}
SPL {X  -165.038, Y  +689.727, Z    +0.000, E1   -11.987, E3 +187425.309}
SPL {X  -165.635, Y  +677.721, Z    +0.000, E1    -3.517, E3 +187424.244}
SPL {X  -165.650, Y  +673.529, Z    +0.000, E1    -0.069, E3 +187423.371}
SPL {X  -165.650, Y  +671.950, Z    +0.000, E1    +1.795, E3 +187422.740}
SPL {X  -165.650, Y  +668.094, Z    +0.000, E1    +7.098, E3 +187422.330}
SPL {X  -165.650, Y  +661.377, Z    +0.000, E1   +18.170, E3 +187422.270}
SPL {X  -165.650, Y  +654.692, Z    +0.000, E1   +29.740, E3 +187421.518}
SPL {X  -165.650, Y  +648.240, Z    +0.000, E1   +42.276, E3 +187417.247}
SPL {X  -165.650, Y  +638.477, Z    +0.000, E1   +48.488, E3 +187423.748}
SPL {X  -165.650, Y  +615.287, Z    +0.000, E1   +74.123, E3 +187408.279}
SPL {X  -165.650, Y  +589.967, Z    +0.000, E1   +71.395, E3 +187424.622}
SPL {X  -165.650, Y  +573.012, Z    +0.000, E1   +68.475, E3 +187440.835}
SPL {X  -165.650, Y  +459.505, Z    +0.000, E1   +68.780, E3 +187512.559}
ENDSPLINE

SPLINE
SPL {X  -165.650, Y  +483.715, Z    +0.000, E1   +63.891, E3 +187528.853}
ENDSPLINE

SPLINE
SPL {X  -165.650, Y  +474.626, Z    +0.000, E1   +63.707, E3 +187539.382}
SPL {X  -165.650, Y  +465.190, Z    +0.000, E1   +63.660, E3 +187549.236}
SPL {X  -165.650, Y  +456.011, Z    +0.000, E1   +63.585, E3 +187559.131}
SPL {X  -165.650, Y  +441.325, Z    +0.000, E1   +63.847, E3 +187572.100}
SPL {X  -165.552, Y  +372.799, Z    +0.000, E1   +69.633, E3 +187584.506}
SPL {X  -165.443, Y  +370.231, Z    +0.000, E1   +68.724, E3 +187594.436}
SPL {X  -164.908, Y  +362.840, Z    +0.000, E1   +68.443, E3 +187602.781}
SPL {X  -164.361, Y  +357.877, Z    +0.000, E1   +67.700, E3 +187613.235}
SPL {X  -163.803, Y  +353.836, Z    +0.000, E1   +66.282, E3 +187628.257}
SPL {X  -162.254, Y  +345.129, Z    +0.000, E1   +65.301, E3 +187643.707}
SPL {X  -158.875, Y  +331.610, Z    +0.000, E1   +64.945, E3 +187658.765}
SPL {X  -154.872, Y  +319.724, Z    +0.000, E1   +64.496, E3 +187672.679}
SPL {X  -152.078, Y  +312.833, Z    +0.000, E1   +64.044, E3 +187681.728}
SPL {X  -149.447, Y  +307.046, Z    +0.000, E1   +63.460, E3 +187690.769}
SPL {X  -145.492, Y  +299.305, Z    +0.000, E1   +63.037, E3 +187700.243}
SPL {X  -142.120, Y  +293.401, Z    +0.000, E1   +62.602, E3 +187707.922}
SPL {X  -139.854, Y  +289.726, Z    +0.000, E1   +61.679, E3 +187715.828}
SPL {X  -135.997, Y  +283.923, Z    +0.000, E1   +62.034, E3 +187719.477}
SPL {X  -124.991, Y  +269.793, Z    +0.000, E1   +65.852, E3 +187714.466}
SPL {X   -80.641, Y  +233.804, Z    +0.000, E1   +55.283, E3 +187845.581}
ENDSPLINE

SPLINE
SPL {X  -126.633, Y  +271.710, Z    +0.000, E1   +51.055, E3 +187976.047}
SPL {X  -147.744, Y  +303.590, Z    +0.000, E1   +42.717, E3 +187984.539}
SPL {X  -158.730, Y  +331.121, Z    +0.000, E1   +31.334, E3 +187984.447}
SPL {X  -162.799, Y  +347.901, Z    +0.000, E1   +22.644, E3 +187987.040}
SPL {X  -164.930, Y  +363.071, Z    +0.000, E1   +13.041, E3 +187984.780}
SPL {X  -165.571, Y  +373.394, Z    +0.000, E1    +5.725, E3 +187985.122}
SPL {X  -165.650, Y  +380.761, Z    +0.000, E1    -0.041, E3 +187983.266}
SPL {X  -165.650, Y  +385.791, Z    +0.000, E1    -7.347, E3 +187982.539}
SPL {X  -165.650, Y  +390.879, Z    +0.000, E1   -16.263, E3 +187981.825}
SPL {X  -165.650, Y  +395.103, Z    +0.000, E1   -23.932, E3 +187981.423}
SPL {X  -165.650, Y  +401.925, Z    +0.000, E1   -35.470, E3 +187980.690}
SPL {X  -165.650, Y  +410.900, Z    +0.000, E1   -46.977, E3 +187981.307}
SPL {X  -165.650, Y  +423.066, Z    +0.000, E1   -61.140, E3 +187977.038}
SPL {X  -165.650, Y  +461.121, Z    +0.000, E1   -74.504, E3 +187978.387}
SPL {X  -165.650, Y  +487.674, Z    +0.000, E1   -70.215, E3 +188001.198}
SPL {X  -165.650, Y  +585.482, Z    +0.000, E1   -67.026, E3 +188080.360}
ENDSPLINE

SPLINE
SPL {X  -165.650, Y  +577.780, Z    +0.000, E1   -64.060, E3 +188096.572}
ENDSPLINE

SPLINE
SPL {X  -165.650, Y  +590.532, Z    +0.000, E1   -63.993, E3 +188109.610}
SPL {X  -165.650, Y  +600.616, Z    +0.000, E1   -64.059, E3 +188119.184}
SPL {X  -165.650, Y  +609.299, Z    +0.000, E1   -64.001, E3 +188128.209}
SPL {X  -165.650, Y  +618.778, Z    +0.000, E1   -63.957, E3 +188138.066}
SPL {X  -165.650, Y  +634.916, Z    +0.000, E1   -64.117, E3 +188153.114}
SPL {X  -165.650, Y  +648.710, Z    +0.000, E1   -63.999, E3 +188167.525}
SPL {X  -165.650, Y  +658.618, Z    +0.000, E1   -64.006, E3 +188177.342}
SPL {X  -165.650, Y  +670.604, Z    +0.000, E1   -64.021, E3 +188189.255}
SPL {X  -165.553, Y  +681.156, Z    +0.000, E1   -63.834, E3 +188201.130}
SPL {X  -164.651, Y  +693.668, Z    +0.000, E1   -63.860, E3 +188213.655}
SPL {X  -162.406, Y  +708.122, Z    +0.000, E1   -63.726, E3 +188228.949}
SPL {X  -159.930, Y  +718.656, Z    +0.000, E1   -63.142, E3 +188243.559}
SPL {X  -156.651, Y  +729.355, Z    +0.000, E1   -62.675, E3 +188257.396}
SPL {X  -153.281, Y  +738.308, Z    +0.000, E1   -62.233, E3 +188268.996}
SPL {X  -150.070, Y  +745.636, Z    +0.000, E1   -61.982, E3 +188277.743}
SPL {X  -148.438, Y  +749.026, Z    +0.000, E1   -61.150, E3 +188285.749}
SPL {X  -145.760, Y  +754.202, Z    +0.000, E1   -61.108, E3 +188291.166}
SPL {X  -143.078, Y  +758.979, Z    +0.000, E1   -60.553, E3 +188298.824}
SPL {X  -139.815, Y  +764.336, Z    +0.000, E1   -60.025, E3 +188306.676}
SPL {X  -133.503, Y  +773.566, Z    +0.000, E1   -62.412, E3 +188304.803}
SPL {X  -122.896, Y  +786.569, Z    +0.000, E1   -64.831, E3 +188304.963}
SPL {X   -84.123, Y  +818.200, Z    +0.000, E1   -55.499, E3 +188418.480}
ENDSPLINE

SPLINE
SPL {X  -127.502, Y  +781.251, Z    +0.000, E1   -49.821, E3 +188550.614}
SPL {X  -156.175, Y  +730.721, Z    +0.000, E1   -34.737, E3 +188566.893}
SPL {X  -163.701, Y  +700.836, Z    +0.000, E1   -18.960, E3 +188563.088}
SPL {X  -165.229, Y  +687.300, Z    +0.000, E1   -10.302, E3 +188563.044}
SPL {X  -165.635, Y  +677.721, Z    +0.000, E1    -3.517, E3 +188562.175}
SPL {X  -165.650, Y  +672.966, Z    +0.000, E1    +0.394, E3 +188561.078}
SPL {X  -165.650, Y  +668.094, Z    +0.000, E1    +7.098, E3 +188560.261}
SPL {X  -165.650, Y  +661.377, Z    +0.000, E1   +18.170, E3 +188560.201}
SPL {X  -165.650, Y  +654.692, Z    +0.000, E1   +29.740, E3 +188559.449}
SPL {X  -165.650, Y  +648.240, Z    +0.000, E1   +42.276, E3 +188555.178}
SPL {X  -165.650, Y  +638.477, Z    +0.000, E1   +48.488, E3 +188561.679}
SPL {X  -165.650, Y  +615.287, Z    +0.000, E1   +74.123, E3 +188546.210}
SPL {X  -165.650, Y  +589.967, Z    +0.000, E1   +71.395, E3 +188562.553}
SPL {X  -165.650, Y  +573.012, Z    +0.000, E1   +68.475, E3 +188578.766}
SPL {X  -165.650, Y  +459.505, Z    +0.000, E1   +68.780, E3 +188650.490}
ENDSPLINE

SPLINE
SPL {X  -165.650, Y  +483.715, Z    +0.000, E1   +63.891, E3 +188666.784}
ENDSPLINE

SPLINE
SPL {X  -165.650, Y  +474.626, Z    +0.000, E1   +63.707, E3 +188677.313}
SPL {X  -165.650, Y  +465.190, Z    +0.000, E1   +63.660, E3 +188687.167}
SPL {X  -165.650, Y  +456.011, Z    +0.000, E1   +63.585, E3 +188697.062}
SPL {X  -165.650, Y  +441.325, Z    +0.000, E1   +63.847, E3 +188710.031}
SPL {X  -165.552, Y  +372.799, Z    +0.000, E1   +69.633, E3 +188722.437}
SPL {X  -165.443, Y  +370.231, Z    +0.000, E1   +68.724, E3 +188732.367}
SPL {X  -164.776, Y  +361.504, Z    +0.000, E1   +68.225, E3 +188743.842}
SPL {X  -164.241, Y  +356.944, Z    +0.000, E1   +66.930, E3 +188758.364}
SPL {X  -163.312, Y  +350.765, Z    +0.000, E1   +66.182, E3 +188769.541}
SPL {X  -163.046, Y  +349.241, Z    +0.000, E1   +65.245, E3 +188778.113}
SPL {X  -160.229, Y  +336.468, Z    +0.000, E1   +65.236, E3 +188790.097}
SPL {X  -157.078, Y  +325.903, Z    +0.000, E1   +64.692, E3 +188803.542}
SPL {X  -153.279, Y  +315.688, Z    +0.000, E1   +64.219, E3 +188816.115}
SPL {X  -149.447, Y  +307.046, Z    +0.000, E1   +63.460, E3 +188828.700}
SPL {X  -145.492, Y  +299.305, Z    +0.000, E1   +63.037, E3 +188838.174}
SPL {X  -142.120, Y  +293.401, Z    +0.000, E1   +62.602, E3 +188845.854}
SPL {X  -139.854, Y  +289.726, Z    +0.000, E1   +61.679, E3 +188853.759}
SPL {X  -135.997, Y  +283.923, Z    +0.000, E1   +62.034, E3 +188857.408}
SPL {X  -124.991, Y  +269.793, Z    +0.000, E1   +65.852, E3 +188852.397}
SPL {X   -80.641, Y  +233.804, Z    +0.000, E1   +55.283, E3 +188983.512}
ENDSPLINE

SPLINE
SPL {X  -126.633, Y  +271.710, Z    +0.000, E1   +51.055, E3 +189113.978}
SPL {X  -147.744, Y  +303.590, Z    +0.000, E1   +42.717, E3 +189122.470}
SPL {X  -158.730, Y  +331.121, Z    +0.000, E1   +31.334, E3 +189122.378}
SPL {X  -162.799, Y  +347.901, Z    +0.000, E1   +22.644, E3 +189124.971}
SPL {X  -164.930, Y  +363.071, Z    +0.000, E1   +13.041, E3 +189122.712}
SPL {X  -165.629, Y  +375.893, Z    +0.000, E1    +3.908, E3 +189122.569}
SPL {X  -165.650, Y  +381.007, Z    +0.000, E1    -0.398, E3 +189121.109}
SPL {X  -165.650, Y  +385.791, Z    +0.000, E1    -7.347, E3 +189120.470}
SPL {X  -165.650, Y  +392.519, Z    +0.000, E1   -19.014, E3 +189119.600}
SPL {X  -165.650, Y  +401.925, Z    +0.000, E1   -35.470, E3 +189118.621}
SPL {X  -165.650, Y  +410.900, Z    +0.000, E1   -46.977, E3 +189119.238}
SPL {X  -165.650, Y  +420.865, Z    +0.000, E1   -58.704, E3 +189116.129}
SPL {X  -165.650, Y  +450.181, Z    +0.000, E1   -73.218, E3 +189114.077}
SPL {X  -165.650, Y  +487.674, Z    +0.000, E1   -70.215, E3 +189139.129}
SPL {X  -165.650, Y  +585.482, Z    +0.000, E1   -67.026, E3 +189218.291}
ENDSPLINE

SPLINE
SPL {X  -165.650, Y  +577.780, Z    +0.000, E1   -64.060, E3 +189234.503}
ENDSPLINE

SPLINE
SPL {X  -165.650, Y  +590.532, Z    +0.000, E1   -63.993, E3 +189247.541}
SPL {X  -165.650, Y  +600.616, Z    +0.000, E1   -64.059, E3 +189257.115}
SPL {X  -165.650, Y  +609.299, Z    +0.000, E1   -64.001, E3 +189266.140}
SPL {X  -165.650, Y  +618.778, Z    +0.000, E1   -63.957, E3 +189275.997}
SPL {X  -165.650, Y  +627.902, Z    +0.000, E1   -63.871, E3 +189285.723}
SPL {X  -165.650, Y  +640.120, Z    +0.000, E1   -64.248, E3 +189295.064}
SPL {X  -165.650, Y  +648.710, Z    +0.000, E1   -63.999, E3 +189305.456}
SPL {X  -165.650, Y  +658.618, Z    +0.000, E1   -64.006, E3 +189315.273}
SPL {X  -165.650, Y  +670.604, Z    +0.000, E1   -64.021, E3 +189327.186}
SPL {X  -165.553, Y  +681.156, Z    +0.000, E1   -63.834, E3 +189339.061}
SPL {X  -164.651, Y  +693.668, Z    +0.000, E1   -63.860, E3 +189351.586}
SPL {X  -163.017, Y  +704.915, Z    +0.000, E1   -63.665, E3 +189364.029}
SPL {X  -161.003, Y  +714.463, Z    +0.000, E1   -63.428, E3 +189375.345}
SPL {X  -157.854, Y  +725.721, Z    +0.000, E1   -62.989, E3 +189389.594}
SPL {X  -155.984, Y  +731.258, Z    +0.000, E1   -62.241, E3 +189399.739}
SPL {X  -153.281, Y  +738.308, Z    +0.000, E1   -62.233, E3 +189406.927}
SPL {X  -150.070, Y  +745.636, Z    +0.000, E1   -61.982, E3 +189415.674}
SPL {X  -146.912, Y  +752.029, Z    +0.000, E1   -61.155, E3 +189426.776}
SPL {X  -143.078, Y  +758.979, Z    +0.000, E1   -60.553, E3 +189436.755}
SPL {X  -139.815, Y  +764.336, Z    +0.000, E1   -60.025, E3 +189444.607}
SPL {X  -133.503, Y  +773.566, Z    +0.000, E1   -62.412, E3 +189442.734}
SPL {X  -122.896, Y  +786.569, Z    +0.000, E1   -64.831, E3 +189442.894}
SPL {X   -84.728, Y  +817.841, Z    +0.000, E1   -56.970, E3 +189533.570}
ENDSPLINE

SPLINE
SPL {X   -85.913, Y  +817.129, Z    +0.000, E1   -53.985, E3 +189589.829}
SPL {X  -116.242, Y  +793.515, Z    +0.000, E1   -51.439, E3 +189674.284}
SPL {X  -136.975, Y  +768.655, Z    +0.000, E1   -47.464, E3 +189698.740}
SPL {X  -151.617, Y  +742.224, Z    +0.000, E1   -39.442, E3 +189705.127}
SPL {X  -159.277, Y  +721.007, Z    +0.000, E1   -30.118, E3 +189704.304}
SPL {X  -163.701, Y  +700.836, Z    +0.000, E1   -18.960, E3 +189701.019}
SPL {X  -165.229, Y  +687.300, Z    +0.000, E1   -10.302, E3 +189700.975}
SPL {X  -165.635, Y  +677.721, Z    +0.000, E1    -3.517, E3 +189700.106}
SPL {X  -165.650, Y  +672.966, Z    +0.000, E1    +0.394, E3 +189699.009}
SPL {X  -165.650, Y  +668.094, Z    +0.000, E1    +7.098, E3 +189698.192}
SPL {X  -165.650, Y  +661.377, Z    +0.000, E1   +18.170, E3 +189698.132}
SPL {X  -165.650, Y  +654.692, Z    +0.000, E1   +29.740, E3 +189697.380}
SPL {X  -165.650, Y  +648.240, Z    +0.000, E1   +42.276, E3 +189693.109}
SPL {X  -165.650, Y  +638.782, Z    +0.000, E1   +47.719, E3 +189700.319}
SPL {X  -165.650, Y  +622.329, Z    +0.000, E1   +68.753, E3 +189687.858}
SPL {X  -165.650, Y  +589.967, Z    +0.000, E1   +71.395, E3 +189700.484}
SPL {X  -165.650, Y  +573.012, Z    +0.000, E1   +68.475, E3 +189716.697}
SPL {X  -165.650, Y  +459.505, Z    +0.000, E1   +68.780, E3 +189788.421}
ENDSPLINE

SPLINE
SPL {X  -165.650, Y  +483.715, Z    +0.000, E1   +63.891, E3 +189804.715}
ENDSPLINE

SPLINE
SPL {X  -165.650, Y  +474.626, Z    +0.000, E1   +63.707, E3 +189815.244}
SPL {X  -165.650, Y  +465.190, Z    +0.000, E1   +63.660, E3 +189825.099}
SPL {X  -165.650, Y  +456.011, Z    +0.000, E1   +63.585, E3 +189834.993}
SPL {X  -165.650, Y  +441.325, Z    +0.000, E1   +63.847, E3 +189847.962}
SPL {X  -165.552, Y  +372.799, Z    +0.000, E1   +69.633, E3 +189860.368}
SPL {X  -165.443, Y  +370.231, Z    +0.000, E1   +68.724, E3 +189870.298}
SPL {X  -164.776, Y  +361.504, Z    +0.000, E1   +68.225, E3 +189881.773}
SPL {X  -164.241, Y  +356.944, Z    +0.000, E1   +66.930, E3 +189896.295}
SPL {X  -163.312, Y  +350.765, Z    +0.000, E1   +66.182, E3 +189907.472}
SPL {X  -163.046, Y  +349.241, Z    +0.000, E1   +65.245, E3 +189916.044}
SPL {X  -160.229, Y  +336.468, Z    +0.000, E1   +65.236, E3 +189928.028}
SPL {X  -157.078, Y  +325.903, Z    +0.000, E1   +64.692, E3 +189941.473}
SPL {X  -153.279, Y  +315.688, Z    +0.000, E1   +64.219, E3 +189954.046}
SPL {X  -149.447, Y  +307.046, Z    +0.000, E1   +63.460, E3 +189966.631}
SPL {X  -145.492, Y  +299.305, Z    +0.000, E1   +63.037, E3 +189976.105}
SPL {X  -142.120, Y  +293.401, Z    +0.000, E1   +62.602, E3 +189983.785}
SPL {X  -139.854, Y  +289.726, Z    +0.000, E1   +61.679, E3 +189991.690}
SPL {X  -135.997, Y  +283.923, Z    +0.000, E1   +62.034, E3 +189995.339}
SPL {X  -124.991, Y  +269.793, Z    +0.000, E1   +65.852, E3 +189990.328}
SPL {X   -80.641, Y  +233.804, Z    +0.000, E1   +55.283, E3 +190121.443}
ENDSPLINE

SPLINE
SPL {X  -126.633, Y  +271.710, Z    +0.000, E1   +51.055, E3 +190251.909}
SPL {X  -147.744, Y  +303.590, Z    +0.000, E1   +42.717, E3 +190260.401}
SPL {X  -158.730, Y  +331.121, Z    +0.000, E1   +31.334, E3 +190260.309}
SPL {X  -162.799, Y  +347.901, Z    +0.000, E1   +22.644, E3 +190262.903}
SPL {X  -164.930, Y  +363.071, Z    +0.000, E1   +13.041, E3 +190260.643}
SPL {X  -165.629, Y  +375.893, Z    +0.000, E1    +3.908, E3 +190260.500}
SPL {X  -165.650, Y  +380.596, Z    +0.000, E1    -0.052, E3 +190259.182}
SPL {X  -165.650, Y  +383.460, Z    +0.000, E1    -3.790, E3 +190258.507}
SPL {X  -165.650, Y  +389.311, Z    +0.000, E1   -13.234, E3 +190257.992}
SPL {X  -165.650, Y  +395.103, Z    +0.000, E1   -23.932, E3 +190257.285}
SPL {X  -165.650, Y  +401.925, Z    +0.000, E1   -35.470, E3 +190256.552}
SPL {X  -165.650, Y  +410.900, Z    +0.000, E1   -46.977, E3 +190257.169}
SPL {X  -165.650, Y  +420.865, Z    +0.000, E1   -58.704, E3 +190254.060}
SPL {X  -165.650, Y  +450.181, Z    +0.000, E1   -73.218, E3 +190252.008}
SPL {X  -165.650, Y  +487.674, Z    +0.000, E1   -70.215, E3 +190277.060}
SPL {X  -165.650, Y  +590.449, Z    +0.000, E1   -68.990, E3 +190345.005}
ENDSPLINE

SPLINE
SPL {X  -165.650, Y  +577.071, Z    +0.000, E1   -65.152, E3 +190363.328}
ENDSPLINE

SPLINE
SPL {X  -165.650, Y  +580.077, Z    +0.000, E1   -64.018, E3 +190374.906}
SPL {X  -165.650, Y  +590.532, Z    +0.000, E1   -63.993, E3 +190385.472}
SPL {X  -165.650, Y  +604.471, Z    +0.000, E1   -64.071, E3 +190398.980}
SPL {X  -165.650, Y  +618.778, Z    +0.000, E1   -63.957, E3 +190413.928}
SPL {X  -165.650, Y  +634.916, Z    +0.000, E1   -64.117, E3 +190428.976}
SPL {X  -165.650, Y  +648.710, Z    +0.000, E1   -63.999, E3 +190443.387}
SPL {X  -165.650, Y  +658.618, Z    +0.000, E1   -64.006, E3 +190453.204}
SPL {X  -165.650, Y  +670.604, Z    +0.000, E1   -64.021, E3 +190465.117}
SPL {X  -165.553, Y  +681.156, Z    +0.000, E1   -63.834, E3 +190476.992}
SPL {X  -164.902, Y  +691.221, Z    +0.000, E1   -64.073, E3 +190485.251}
SPL {X  -163.641, Y  +701.218, Z    +0.000, E1   -63.638, E3 +190498.604}
SPL {X  -161.003, Y  +714.463, Z    +0.000, E1   -63.428, E3 +190513.276}
SPL {X  -158.978, Y  +722.038, Z    +0.000, E1   -63.038, E3 +190523.343}
SPL {X  -156.651, Y  +729.355, Z    +0.000, E1   -62.675, E3 +190533.258}
SPL {X  -153.281, Y  +738.308, Z    +0.000, E1   -62.233, E3 +190544.858}
SPL {X  -150.070, Y  +745.636, Z    +0.000, E1   -61.982, E3 +190553.605}
SPL {X  -146.912, Y  +752.029, Z    +0.000, E1   -61.155, E3 +190564.707}
SPL {X  -143.078, Y  +758.979, Z    +0.000, E1   -60.553, E3 +190574.686}
SPL {X  -139.815, Y  +764.336, Z    +0.000, E1   -60.025, E3 +190582.538}
SPL {X  -130.672, Y  +777.307, Z    +0.000, E1   -63.098, E3 +190580.829}
SPL {X   -84.123, Y  +818.200, Z    +0.000, E1   -55.499, E3 +190694.342}
ENDSPLINE

SPLINE
SPL {X  -127.502, Y  +781.251, Z    +0.000, E1   -49.821, E3 +190826.476}
SPL {X  -156.175, Y  +730.721, Z    +0.000, E1   -34.737, E3 +190842.755}
SPL {X  -163.701, Y  +700.836, Z    +0.000, E1   -18.960, E3 +190838.950}
SPL {X  -165.229, Y  +687.300, Z    +0.000, E1   -10.302, E3 +190838.906}
SPL {X  -165.635, Y  +677.721, Z    +0.000, E1    -3.517, E3 +190838.037}
SPL {X  -165.650, Y  +672.966, Z    +0.000, E1    +0.394, E3 +190836.940}
SPL {X  -165.650, Y  +668.094, Z    +0.000, E1    +7.098, E3 +190836.123}
SPL {X  -165.650, Y  +662.291, Z    +0.000, E1   +16.729, E3 +190836.048}
SPL {X  -165.650, Y  +656.382, Z    +0.000, E1   +26.732, E3 +190835.606}
SPL {X  -165.650, Y  +648.240, Z    +0.000, E1   +42.276, E3 +190831.040}
SPL {X  -165.650, Y  +638.477, Z    +0.000, E1   +48.488, E3 +190837.541}
SPL {X  -165.650, Y  +615.287, Z    +0.000, E1   +74.123, E3 +190822.072}
SPL {X  -165.650, Y  +589.967, Z    +0.000, E1   +71.395, E3 +190838.415}
SPL {X  -165.650, Y  +573.012, Z    +0.000, E1   +68.475, E3 +190854.628}
SPL {X  -165.650, Y  +459.505, Z    +0.000, E1   +68.780, E3 +190926.352}
ENDSPLINE

SPLINE
SPL {X  -165.650, Y  +483.715, Z    +0.000, E1   +63.891, E3 +190942.646}
ENDSPLINE

SPLINE
SPL {X  -165.650, Y  +474.626, Z    +0.000, E1   +63.707, E3 +190953.175}
SPL {X  -165.650, Y  +465.190, Z    +0.000, E1   +63.660, E3 +190963.030}
SPL {X  -165.650, Y  +456.011, Z    +0.000, E1   +63.585, E3 +190972.924}
SPL {X  -165.650, Y  +441.325, Z    +0.000, E1   +63.847, E3 +190985.894}
SPL {X  -165.552, Y  +372.799, Z    +0.000, E1   +69.633, E3 +190998.299}
SPL {X  -165.188, Y  +366.130, Z    +0.000, E1   +68.611, E3 +191012.702}
SPL {X  -164.361, Y  +357.877, Z    +0.000, E1   +67.700, E3 +191027.029}
SPL {X  -164.353, Y  +357.815, Z    +0.000, E1   +66.333, E3 +191037.930}
SPL {X  -163.312, Y  +350.765, Z    +0.000, E1   +66.182, E3 +191045.403}
SPL {X  -163.046, Y  +349.241, Z    +0.000, E1   +65.245, E3 +191053.975}
SPL {X  -160.229, Y  +336.468, Z    +0.000, E1   +65.236, E3 +191065.959}
SPL {X  -158.158, Y  +329.247, Z    +0.000, E1   +64.622, E3 +191076.730}
SPL {X  -154.872, Y  +319.724, Z    +0.000, E1   +64.496, E3 +191086.473}
SPL {X  -151.091, Y  +310.592, Z    +0.000, E1   +63.929, E3 +191098.412}
SPL {X  -148.836, Y  +305.783, Z    +0.000, E1   +63.120, E3 +191107.544}
SPL {X  -145.492, Y  +299.305, Z    +0.000, E1   +63.037, E3 +191114.036}
SPL {X  -142.120, Y  +293.401, Z    +0.000, E1   +62.602, E3 +191121.716}
SPL {X  -139.854, Y  +289.726, Z    +0.000, E1   +61.679, E3 +191129.621}
SPL {X  -135.997, Y  +283.923, Z    +0.000, E1   +62.034, E3 +191133.270}
SPL {X  -124.991, Y  +269.793, Z    +0.000, E1   +65.852, E3 +191128.259}
SPL {X   -80.641, Y  +233.804, Z    +0.000, E1   +55.283, E3 +191259.374}
ENDSPLINE

SPLINE
SPL {X  -132.197, Y  +278.681, Z    +0.000, E1   +49.692, E3 +191393.247}
SPL {X  -156.075, Y  +322.998, Z    +0.000, E1   +35.140, E3 +191398.328}
SPL {X  -163.642, Y  +352.786, Z    +0.000, E1   +19.725, E3 +191400.107}
SPL {X  -165.477, Y  +370.931, Z    +0.000, E1    +7.630, E3 +191398.695}
SPL {X  -165.650, Y  +378.219, Z    +0.000, E1    +1.951, E3 +191397.968}
SPL {X  -165.650, Y  +380.596, Z    +0.000, E1    -0.052, E3 +191397.113}
SPL {X  -165.650, Y  +383.460, Z    +0.000, E1    -3.790, E3 +191396.438}
SPL {X  -165.650, Y  +387.326, Z    +0.000, E1   -10.041, E3 +191396.309}
SPL {X  -165.650, Y  +392.519, Z    +0.000, E1   -19.014, E3 +191395.462}
SPL {X  -165.650, Y  +401.925, Z    +0.000, E1   -35.470, E3 +191394.483}
SPL {X  -165.650, Y  +410.900, Z    +0.000, E1   -46.977, E3 +191395.100}
SPL {X  -165.650, Y  +420.865, Z    +0.000, E1   -58.704, E3 +191391.991}
SPL {X  -165.650, Y  +450.181, Z    +0.000, E1   -73.218, E3 +191389.939}
SPL {X  -165.650, Y  +487.674, Z    +0.000, E1   -70.215, E3 +191414.991}
SPL {X  -165.650, Y  +590.449, Z    +0.000, E1   -68.990, E3 +191482.936}
ENDSPLINE

SPLINE
SPL {X  -165.650, Y  +577.071, Z    +0.000, E1   -65.152, E3 +191501.259}
ENDSPLINE

SPLINE
SPL {X  -165.650, Y  +580.077, Z    +0.000, E1   -64.018, E3 +191512.837}
SPL {X  -165.650, Y  +590.532, Z    +0.000, E1   -63.993, E3 +191523.403}
SPL {X  -165.650, Y  +604.471, Z    +0.000, E1   -64.071, E3 +191536.911}
SPL {X  -165.650, Y  +618.778, Z    +0.000, E1   -63.957, E3 +191551.859}
SPL {X  -165.650, Y  +627.902, Z    +0.000, E1   -63.871, E3 +191561.585}
SPL {X  -165.650, Y  +640.120, Z    +0.000, E1   -64.248, E3 +191570.926}
SPL {X  -165.650, Y  +648.710, Z    +0.000, E1   -63.999, E3 +191581.318}
SPL {X  -165.650, Y  +660.990, Z    +0.000, E1   -63.976, E3 +191593.843}
SPL {X  -165.633, Y  +677.852, Z    +0.000, E1   -63.999, E3 +191610.616}
SPL {X  -164.651, Y  +693.668, Z    +0.000, E1   -63.860, E3 +191627.448}
SPL {X  -162.406, Y  +708.122, Z    +0.000, E1   -63.726, E3 +191642.742}
SPL {X  -159.930, Y  +718.656, Z    +0.000, E1   -63.142, E3 +191657.353}
SPL {X  -156.651, Y  +729.355, Z    +0.000, E1   -62.675, E3 +191671.189}
SPL {X  -153.281, Y  +738.308, Z    +0.000, E1   -62.233, E3 +191682.789}
SPL {X  -150.070, Y  +745.636, Z    +0.000, E1   -61.982, E3 +191691.536}
SPL {X  -148.438, Y  +749.026, Z    +0.000, E1   -61.150, E3 +191699.542}
SPL {X  -145.760, Y  +754.202, Z    +0.000, E1   -61.108, E3 +191704.959}
SPL {X  -143.078, Y  +758.979, Z    +0.000, E1   -60.553, E3 +191712.618}
SPL {X  -139.815, Y  +764.336, Z    +0.000, E1   -60.025, E3 +191720.469}
SPL {X  -130.672, Y  +777.307, Z    +0.000, E1   -63.098, E3 +191718.760}
SPL {X   -84.123, Y  +818.200, Z    +0.000, E1   -55.499, E3 +191832.274}
ENDSPLINE

SPLINE
SPL {X  -127.502, Y  +781.251, Z    +0.000, E1   -49.821, E3 +191964.407}
SPL {X  -151.617, Y  +742.224, Z    +0.000, E1   -39.442, E3 +191980.989}
SPL {X  -159.277, Y  +721.007, Z    +0.000, E1   -30.118, E3 +191980.167}
SPL {X  -163.701, Y  +700.836, Z    +0.000, E1   -18.960, E3 +191976.881}
SPL {X  -165.229, Y  +687.300, Z    +0.000, E1   -10.302, E3 +191976.837}
SPL {X  -165.592, Y  +679.896, Z    +0.000, E1    -5.071, E3 +191976.117}
SPL {X  -165.650, Y  +674.350, Z    +0.000, E1    -0.828, E3 +191975.491}
SPL {X  -165.650, Y  +672.653, Z    +0.000, E1    +0.827, E3 +191974.684}
SPL {X  -165.650, Y  +668.094, Z    +0.000, E1    +7.098, E3 +191974.054}
SPL {X  -165.650, Y  +662.291, Z    +0.000, E1   +16.729, E3 +191973.979}
SPL {X  -165.650, Y  +656.382, Z    +0.000, E1   +26.732, E3 +191973.537}
SPL {X  -165.650, Y  +648.240, Z    +0.000, E1   +42.276, E3 +191968.971}
SPL {X  -165.650, Y  +638.782, Z    +0.000, E1   +47.719, E3 +191976.181}
SPL {X  -165.650, Y  +622.329, Z    +0.000, E1   +68.753, E3 +191963.720}
SPL {X  -165.650, Y  +589.967, Z    +0.000, E1   +71.395, E3 +191976.346}
SPL {X  -165.650, Y  +573.012, Z    +0.000, E1   +68.475, E3 +191992.559}
SPL {X  -165.650, Y  +459.505, Z    +0.000, E1   +68.780, E3 +192064.283}
ENDSPLINE

SPLINE
SPL {X  -165.650, Y  +483.715, Z    +0.000, E1   +63.891, E3 +192080.577}
ENDSPLINE

SPLINE
SPL {X  -165.650, Y  +474.626, Z    +0.000, E1   +63.707, E3 +192091.106}
SPL {X  -165.650, Y  +465.190, Z    +0.000, E1   +63.660, E3 +192100.961}
SPL {X  -165.650, Y  +456.011, Z    +0.000, E1   +63.585, E3 +192110.855}
SPL {X  -165.650, Y  +441.325, Z    +0.000, E1   +63.847, E3 +192123.825}
SPL {X  -165.552, Y  +372.799, Z    +0.000, E1   +69.633, E3 +192136.230}
SPL {X  -165.443, Y  +370.231, Z    +0.000, E1   +68.724, E3 +192146.160}
SPL {X  -164.776, Y  +361.504, Z    +0.000, E1   +68.225, E3 +192157.635}
SPL {X  -164.137, Y  +356.163, Z    +0.000, E1   +67.495, E3 +192167.925}
SPL {X  -163.803, Y  +353.836, Z    +0.000, E1   +66.282, E3 +192179.981}
SPL {X  -162.254, Y  +345.129, Z    +0.000, E1   +65.301, E3 +192195.431}
SPL {X  -159.503, Y  +333.793, Z    +0.000, E1   +65.139, E3 +192206.875}
SPL {X  -157.078, Y  +325.903, Z    +0.000, E1   +64.692, E3 +192217.335}
SPL {X  -153.279, Y  +315.688, Z    +0.000, E1   +64.219, E3 +192229.908}
SPL {X  -149.447, Y  +307.046, Z    +0.000, E1   +63.460, E3 +192242.493}
SPL {X  -145.492, Y  +299.305, Z    +0.000, E1   +63.037, E3 +192251.967}
SPL {X  -142.120, Y  +293.401, Z    +0.000, E1   +62.602, E3 +192259.647}
SPL {X  -139.854, Y  +289.726, Z    +0.000, E1   +61.679, E3 +192267.552}
SPL {X  -135.997, Y  +283.923, Z    +0.000, E1   +62.034, E3 +192271.201}
SPL {X  -124.991, Y  +269.793, Z    +0.000, E1   +65.852, E3 +192266.191}
SPL {X   -80.641, Y  +233.804, Z    +0.000, E1   +55.283, E3 +192397.305}
ENDSPLINE

SPLINE
SPL {X  -132.197, Y  +278.681, Z    +0.000, E1   +49.692, E3 +192531.178}
SPL {X  -156.075, Y  +322.998, Z    +0.000, E1   +35.140, E3 +192536.259}
SPL {X  -162.799, Y  +347.901, Z    +0.000, E1   +22.644, E3 +192538.765}
SPL {X  -164.930, Y  +363.071, Z    +0.000, E1   +13.041, E3 +192536.505}
SPL {X  -165.629, Y  +375.893, Z    +0.000, E1    +3.908, E3 +192536.362}
SPL {X  -165.650, Y  +380.596, Z    +0.000, E1    -0.052, E3 +192535.044}
SPL {X  -165.650, Y  +383.460, Z    +0.000, E1    -3.790, E3 +192534.369}
SPL {X  -165.650, Y  +389.311, Z    +0.000, E1   -13.234, E3 +192533.854}
SPL {X  -165.650, Y  +395.103, Z    +0.000, E1   -23.932, E3 +192533.147}
SPL {X  -165.650, Y  +401.925, Z    +0.000, E1   -35.470, E3 +192532.414}
SPL {X  -165.650, Y  +410.900, Z    +0.000, E1   -46.977, E3 +192533.031}
SPL {X  -165.650, Y  +420.865, Z    +0.000, E1   -58.704, E3 +192529.922}
SPL {X  -165.650, Y  +450.181, Z    +0.000, E1   -73.218, E3 +192527.870}
SPL {X  -165.650, Y  +487.674, Z    +0.000, E1   -70.215, E3 +192552.922}
SPL {X  -165.650, Y  +590.449, Z    +0.000, E1   -68.990, E3 +192620.867}
ENDSPLINE

SPLINE
SPL {X  -165.650, Y  +577.071, Z    +0.000, E1   -65.152, E3 +192639.190}
ENDSPLINE

